KUKA KRL program: EPS_2_251455_MH61A_A_20251003045103.src

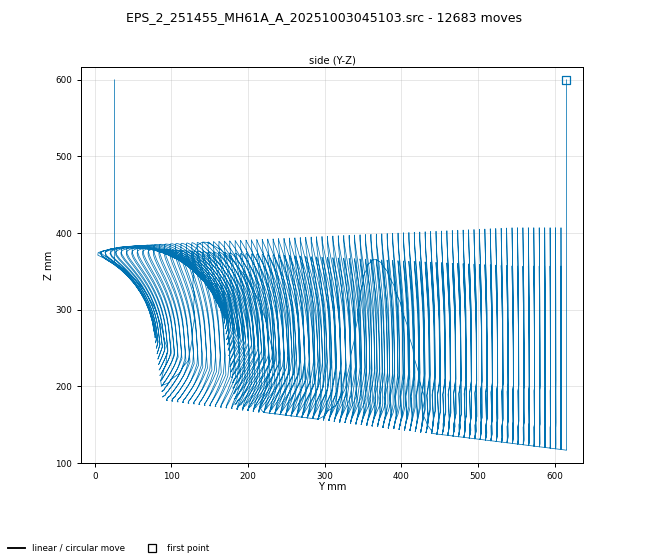
[picture p0: tool path of EPS_2_251455_MH61A_A_20251003045103.src, 12683 of 12685 moves have a stored position in this frame; points joined in program order, loops and branches not executed]
&ACCESS RVP
&REL 4
&COMMENT QRS 19112012
&PARAM EDITMASK = *
DEF PART()
EXT BAS (BAS_COMMAND :IN,REAL :IN )
INT I
BAS (#INITMOV,0 )

;KUKA QRS Post kuka4.cps  Date:22-06-2017 !

File_ID=2871

QRS_PRE_INIT()

;Init var - Until changes are made in qrs_pre_init
Outlet_Square_prg=0
Inlet_1_Square_prg=0
Inlet_2_Square_prg=0
Inlet_3_Square_prg=0
Inlet_4_Square_prg=0
Inlet_5_Square_prg=0

Outlet_1={X 0.000, Y 546.330, Z 306.500, B 0.000, E1 0.000 }
Inlet_1={X 0.000, Y 549.890, Z 256.500, B 0.000, E1 200.000 }
Outlet_1_type=201
Inlet_1_type=201
;QRS#1=Sidecore dimensions
;QRS#2=200-8" PVC SDR 35
;QRS#3=200-8" PVC SDR 35
;QRS#4=
;QRS#5=
;QRS#6=
;QRS#7=
;QRS#8=
;QRS#9=12-08 PSX
;QRS#10=12-08 PSX
;QRS#11=
;QRS#12=
;QRS#13=
;QRS#14=
;QRS#15=
;QRS#16=1220x127x686 2,25'
;QRS#17=EPS Height
;QRS#18=407
;QRS#19=*
;QRS#20= UPDATED VERSION 22-06-2017
;QRS#21=*
Outlet_Square=0100
Inlet_1_Square=0100
Inlet_2_Square=0
Inlet_3_Square=0
Inlet_4_Square=0
Inlet_5_Square=0
Mill_Square=1
Outlet_Square_Prg=204
Inlet_1_Square_prg=204

QRS_INIT()

$ADVANCE=5

; T1
PTP {E1 173.605,E2 173.605}
PTP {X 0,Y 615.512,A -85,B 0,C 180,E1 173.605,E2 173.605,E3 0,E4 0,E5 0,E6 0}
QRS_SPEED_INIT()
LIN {X 0,Y 615.512,Z 600,A -85,B 0,C 180,E1 173.605,E2 173.605,E3 0,E4 0,E5 0,E6 0} C_VEL
LIN {X 0,Y 615.512,Z 126.872,A -85,B 0,C 180,E1 173.605,E2 173.605} C_VEL
LIN {X 0,Y 615.512,Z 118.701,A -85,B 0,C 180,E1 173.605,E2 173.605} C_VEL
LIN {X 0,Y 615.489,Z 116.701,A -85,B 0,C 180,E1 173.42,E2 173.42} C_VEL
LIN {X 0,Y 615.462,Z 116.69,A -85,B 0,C 180,E1 170.801,E2 170.801} C_VEL
LIN {X 0,Y 615.487,Z 116.687,A -85,B 0,C 180,E1 168.139,E2 168.139} C_VEL
LIN {X 0,Y 615.481,Z 116.697,A -85,B 0,C 180,E1 165.451,E2 165.451} C_VEL
LIN {X 0,Y 615.47,Z 116.687,A -85,B 0,C 180,E1 162.729,E2 162.729} C_VEL
LIN {X 0,Y 615.49,Z 116.695,A -85,B 0,C 180,E1 159.967,E2 159.967} C_VEL
LIN {X 0,Y 615.479,Z 116.699,A -85,B 0,C 180,E1 157.656,E2 157.656} C_VEL
LIN {X 0,Y 615.464,Z 116.688,A -85,B 0,C 180,E1 155.007,E2 155.007} C_VEL
LIN {X 0,Y 615.489,Z 116.698,A -85,B 0,C 180,E1 152.085,E2 152.085} C_VEL
LIN {X 0,Y 615.484,Z 116.698,A -85,B 0,C 180,E1 149.84,E2 149.84} C_VEL
LIN {X 0,Y 615.463,Z 116.693,A -85,B 0,C 180,E1 147.541,E2 147.541} C_VEL
LIN {X 0,Y 615.466,Z 116.688,A -85,B 0,C 180,E1 145.184,E2 145.184} C_VEL
LIN {X 0,Y 615.495,Z 116.684,A -85,B 0,C 180,E1 142.758,E2 142.758} C_VEL
LIN {X 0,Y 615.472,Z 116.696,A -85,B 0,C 180,E1 139.913,E2 139.913} C_VEL
LIN {X 0,Y 615.458,Z 116.692,A -85,B 0,C 180,E1 137.645,E2 137.645} C_VEL
LIN {X 0,Y 615.496,Z 116.684,A -85,B 0,C 180,E1 134.932,E2 134.932} C_VEL
LIN {X 0,Y 615.471,Z 116.696,A -85,B 0,C 180,E1 132.079,E2 132.079} C_VEL
LIN {X 0,Y 615.459,Z 116.691,A -85,B 0,C 180,E1 129.752,E2 129.752} C_VEL
LIN {X 0,Y 615.491,Z 116.689,A -85,B 0,C 180,E1 126.937,E2 126.937} C_VEL
LIN {X 0,Y 615.459,Z 116.693,A -85,B 0,C 180,E1 124.024,E2 124.024} C_VEL
LIN {X 0,Y 615.464,Z 116.688,A -85,B 0,C 180,E1 121.687,E2 121.687} C_VEL
LIN {X 0,Y 615.486,Z 116.685,A -85,B 0,C 180,E1 119.406,E2 119.406} C_VEL
LIN {X 0,Y 615.471,Z 116.696,A -85,B 0,C 180,E1 116.445,E2 116.445} C_VEL
LIN {X 0,Y 615.461,Z 116.689,A -85,B 0,C 180,E1 114.003,E2 114.003} C_VEL
LIN {X 0,Y 615.496,Z 116.685,A -85,B 0,C 180,E1 111.431,E2 111.431} C_VEL
LIN {X 0,Y 615.469,Z 116.696,A -85,B 0,C 180,E1 108.6,E2 108.6} C_VEL
LIN {X 0,Y 615.475,Z 116.686,A -85,B 0,C 180,E1 105.905,E2 105.905} C_VEL
LIN {X 0,Y 615.491,Z 116.697,A -85,B 0,C 180,E1 103.201,E2 103.201} C_VEL
LIN {X 0,Y 615.46,Z 116.692,A -85,B 0,C 180,E1 100.527,E2 100.527} C_VEL
LIN {X 0,Y 615.485,Z 116.685,A -85,B 0,C 180,E1 97.876,E2 97.876} C_VEL
LIN {X 0,Y 615.494,Z 116.701,A -85,B 0,C 180,E1 95.241,E2 95.241} C_VEL
LIN {X 0,Y 615.459,Z 116.691,A -85,B 0,C 180,E1 92.618,E2 92.618} C_VEL
LIN {X 0,Y 615.486,Z 116.686,A -85,B 0,C 180,E1 90,E2 90} C_VEL
LIN {X 0,Y 615.496,Z 116.879,A -85,B 0,C 180,E1 87.955,E2 87.955} C_VEL
LIN {X 0,Y 615.461,Z 131.384,A -85,B 0,C 180,E1 85.415,E2 85.415} C_VEL
LIN {X 0,Y 615.445,Z 146.098,A -85,B 0,C 180,E1 82.866,E2 82.866} C_VEL
LIN {X 0,Y 615.45,Z 146.551,A -85,B 0,C 180,E1 82.804,E2 82.804} C_VEL
LIN {X 0,Y 615.45,Z 252.819,A -85,B 0,C 180,E1 81.545,E2 81.545} C_VEL
LIN {X 0,Y 615.452,Z 266.001,A -85,B 0,C 180,E1 81.256,E2 81.256} C_VEL
LIN {X 0,Y 615.481,Z 278.61,A -85,B 0,C 180,E1 80.842,E2 80.842} C_VEL
LIN {X 0,Y 615.493,Z 290.7,A -85,B 0,C 180,E1 80.304,E2 80.304} C_VEL
LIN {X 0,Y 615.485,Z 302.179,A -85,B 0,C 180,E1 79.639,E2 79.639} C_VEL
LIN {X 0,Y 615.499,Z 311.681,A -85,B 0,C 180,E1 78.957,E2 78.957} C_VEL
LIN {X 0,Y 615.497,Z 321.042,A -85,B 0,C 180,E1 78.139,E2 78.139} C_VEL
LIN {X 0,Y 615.498,Z 330.259,A -85,B 0,C 180,E1 77.135,E2 77.135} C_VEL
LIN {X 0,Y 615.496,Z 338.117,A -85,B 0,C 180,E1 76.064,E2 76.064} C_VEL
LIN {X 0,Y 615.497,Z 343.66,A -85,B 0,C 180,E1 75.113,E2 75.113} C_VEL
LIN {X 0,Y 615.492,Z 348.346,A -85,B 0,C 180,E1 74.095,E2 74.095} C_VEL
LIN {X 0,Y 615.495,Z 351.892,A -85,B 0,C 180,E1 73.072,E2 73.072} C_VEL
LIN {X 0,Y 615.498,Z 354.389,A -85,B 0,C 180,E1 72.043,E2 72.043} C_VEL
LIN {X 0,Y 615.494,Z 355.474,A -85,B 0,C 180,E1 71.354,E2 71.354} C_VEL
LIN {X 0,Y 615.496,Z 356.136,A -85,B 0,C 180,E1 70.662,E2 70.662} C_VEL
LIN {X 0,Y 615.497,Z 356.267,A -85,B 0,C 180,E1 69.441,E2 69.441} C_VEL
LIN {X 0,Y 615.498,Z 355.487,A -85,B 0,C 180,E1 68.568,E2 68.568} C_VEL
LIN {X 0,Y 615.492,Z 353.93,A -85,B 0,C 180,E1 67.653,E2 67.653} C_VEL
LIN {X 0,Y 615.496,Z 350.636,A -85,B 0,C 180,E1 66.444,E2 66.444} C_VEL
LIN {X 0,Y 615.495,Z 346.435,A -85,B 0,C 180,E1 65.369,E2 65.369} C_VEL
LIN {X 0,Y 615.494,Z 340.815,A -85,B 0,C 180,E1 64.284,E2 64.284} C_VEL
LIN {X 0,Y 615.498,Z 334,A -85,B 0,C 180,E1 63.255,E2 63.255} C_VEL
LIN {X 0,Y 615.499,Z 325.884,A -85,B 0,C 180,E1 62.27,E2 62.27} C_VEL
LIN {X 0,Y 615.497,Z 317.556,A -85,B 0,C 180,E1 61.445,E2 61.445} C_VEL
LIN {X 0,Y 615.498,Z 306.914,A -85,B 0,C 180,E1 60.594,E2 60.594} C_VEL
LIN {X 0,Y 615.46,Z 296.655,A -85,B 0,C 180,E1 59.931,E2 59.931} C_VEL
LIN {X 0,Y 615.489,Z 284.671,A -85,B 0,C 180,E1 59.318,E2 59.318} C_VEL
LIN {X 0,Y 615.495,Z 272.133,A -85,B 0,C 180,E1 58.838,E2 58.838} C_VEL
LIN {X 0,Y 615.481,Z 259.797,A -85,B 0,C 180,E1 58.501,E2 58.501} C_VEL
LIN {X 0,Y 615.471,Z 246.219,A -85,B 0,C 180,E1 58.273,E2 58.273} C_VEL
LIN {X 0,Y 615.485,Z 146.442,A -85,B 0,C 180,E1 57.105,E2 57.105} C_VEL
LIN {X 0,Y 615.488,Z 129.487,A -85,B 0,C 180,E1 54.166,E2 54.166} C_VEL
LIN {X 0,Y 615.444,Z 116.696,A -85,B 0,C 180,E1 51.902,E2 51.902} C_VEL
LIN {X 0,Y 615.449,Z 116.693,A -85,B 0,C 180,E1 49.39,E2 49.39} C_VEL
LIN {X 0,Y 615.498,Z 116.697,A -85,B 0,C 180,E1 46.756,E2 46.756} C_VEL
LIN {X 0,Y 615.441,Z 116.697,A -85,B 0,C 180,E1 44.154,E2 44.154} C_VEL
LIN {X 0,Y 615.434,Z 116.697,A -85,B 0,C 180,E1 42.074,E2 42.074} C_VEL
LIN {X 0,Y 615.434,Z 116.695,A -85,B 0,C 180,E1 39.754,E2 39.754} C_VEL
LIN {X 0,Y 615.487,Z 116.694,A -85,B 0,C 180,E1 37.242,E2 37.242} C_VEL
LIN {X 0,Y 615.455,Z 116.699,A -85,B 0,C 180,E1 34.696,E2 34.696} C_VEL
LIN {X 0,Y 615.427,Z 116.698,A -85,B 0,C 180,E1 32.322,E2 32.322} C_VEL
LIN {X 0,Y 615.444,Z 116.696,A -85,B 0,C 180,E1 29.787,E2 29.787} C_VEL
LIN {X 0,Y 615.466,Z 116.7,A -85,B 0,C 180,E1 27.041,E2 27.041} C_VEL
LIN {X 0,Y 615.452,Z 116.699,A -85,B 0,C 180,E1 24.993,E2 24.993} C_VEL
LIN {X 0,Y 615.431,Z 116.7,A -85,B 0,C 180,E1 22.847,E2 22.847} C_VEL
LIN {X 0,Y 615.417,Z 116.699,A -85,B 0,C 180,E1 20.539,E2 20.539} C_VEL
LIN {X 0,Y 615.449,Z 116.699,A -85,B 0,C 180,E1 17.958,E2 17.958} C_VEL
LIN {X 0,Y 615.442,Z 116.7,A -85,B 0,C 180,E1 15.227,E2 15.227} C_VEL
LIN {X 0,Y 615.434,Z 116.7,A -85,B 0,C 180,E1 13.202,E2 13.202} C_VEL
LIN {X 0,Y 615.415,Z 116.7,A -85,B 0,C 180,E1 10.852,E2 10.852} C_VEL
LIN {X 0,Y 615.424,Z 116.7,A -85,B 0,C 180,E1 8.537,E2 8.537} C_VEL
LIN {X 0,Y 615.498,Z 116.699,A -85,B 0,C 180,E1 5.898,E2 5.898} C_VEL
LIN {X 0,Y 615.428,Z 116.698,A -85,B 0,C 180,E1 3.273,E2 3.273} C_VEL
LIN {X 0,Y 615.428,Z 116.698,A -85,B 0,C 180,E1 1.309,E2 1.309} C_VEL
LIN {X 0,Y 615.429,Z 116.697,A -85,B 0,C 180,E1 -0.654,E2 -0.654} C_VEL
LIN {X 0,Y 615.429,Z 116.697,A -85,B 0,C 180,E1 -2.618,E2 -2.618} C_VEL
LIN {X 0,Y 615.43,Z 116.696,A -85,B 0,C 180,E1 -4.585,E2 -4.585} C_VEL
LIN {X 0,Y 615.431,Z 116.696,A -85,B 0,C 180,E1 -6.557,E2 -6.557} C_VEL
LIN {X 0,Y 615.431,Z 116.696,A -85,B 0,C 180,E1 -8.538,E2 -8.538} C_VEL
LIN {X 0,Y 615.434,Z 116.697,A -85,B 0,C 180,E1 -10.861,E2 -10.861} C_VEL
LIN {X 0,Y 615.465,Z 116.699,A -85,B 0,C 180,E1 -13.202,E2 -13.202} C_VEL
LIN {X 0,Y 615.467,Z 116.692,A -85,B 0,C 180,E1 -15.906,E2 -15.906} C_VEL
LIN {X 0,Y 615.457,Z 116.693,A -85,B 0,C 180,E1 -17.958,E2 -17.958} C_VEL
LIN {X 0,Y 615.439,Z 116.696,A -85,B 0,C 180,E1 -20.544,E2 -20.544} C_VEL
LIN {X 0,Y 615.462,Z 116.698,A -85,B 0,C 180,E1 -22.846,E2 -22.846} C_VEL
LIN {X 0,Y 615.466,Z 116.691,A -85,B 0,C 180,E1 -25.717,E2 -25.717} C_VEL
LIN {X 0,Y 615.448,Z 116.692,A -85,B 0,C 180,E1 -27.917,E2 -27.917} C_VEL
LIN {X 0,Y 615.443,Z 116.694,A -85,B 0,C 180,E1 -30.163,E2 -30.163} C_VEL
LIN {X 0,Y 615.458,Z 116.697,A -85,B 0,C 180,E1 -32.459,E2 -32.459} C_VEL
LIN {X 0,Y 615.499,Z 116.7,A -85,B 0,C 180,E1 -34.815,E2 -34.815} C_VEL
LIN {X 0,Y 615.489,Z 116.687,A -85,B 0,C 180,E1 -37.242,E2 -37.242} C_VEL
LIN {X 0,Y 615.448,Z 116.692,A -85,B 0,C 180,E1 -39.753,E2 -39.753} C_VEL
LIN {X 0,Y 615.477,Z 116.698,A -85,B 0,C 180,E1 -42.354,E2 -42.354} C_VEL
LIN {X 0,Y 615.492,Z 116.685,A -85,B 0,C 180,E1 -45.068,E2 -45.068} C_VEL
LIN {X 0,Y 615.453,Z 116.692,A -85,B 0,C 180,E1 -47.644,E2 -47.644} C_VEL
LIN {X 0,Y 615.493,Z 116.699,A -85,B 0,C 180,E1 -50.25,E2 -50.25} C_VEL
LIN {X 0,Y 615.475,Z 116.686,A -85,B 0,C 180,E1 -53.065,E2 -53.065} C_VEL
LIN {X 0,Y 615.46,Z 116.69,A -85,B 0,C 180,E1 -55.303,E2 -55.303} C_VEL
LIN {X 0,Y 615.464,Z 116.695,A -85,B 0,C 180,E1 -57.673,E2 -57.673} C_VEL
LIN {X 0,Y 615.489,Z 116.686,A -85,B 0,C 180,E1 -60.594,E2 -60.594} C_VEL
LIN {X 0,Y 615.468,Z 116.687,A -85,B 0,C 180,E1 -62.959,E2 -62.959} C_VEL
LIN {X 0,Y 615.485,Z 116.7,A -85,B 0,C 180,E1 -65.728,E2 -65.728} C_VEL
LIN {X 0,Y 615.464,Z 116.822,A -85,B 0,C 180,E1 -67.066,E2 -67.066} C_VEL
LIN {X 0,Y 615.465,Z 136.77,A -85,B 0,C 180,E1 -69.706,E2 -69.706} C_VEL
LIN {X 0,Y 615.485,Z 158.669,A -85,B 0,C 180,E1 -72.558,E2 -72.558} C_VEL
LIN {X 0,Y 615.469,Z 179.891,A -85,B 0,C 180,E1 -75.281,E2 -75.281} C_VEL
LIN {X 0,Y 615.452,Z 194.3,A -85,B 0,C 180,E1 -77.113,E2 -77.113} C_VEL
LIN {X 0,Y 615.488,Z 302.823,A -85,B 0,C 180,E1 -78.411,E2 -78.411} C_VEL
LIN {X 0,Y 615.477,Z 315.341,A -85,B 0,C 180,E1 -78.682,E2 -78.682} C_VEL
LIN {X 0,Y 615.488,Z 328.618,A -85,B 0,C 180,E1 -79.113,E2 -79.113} C_VEL
LIN {X 0,Y 615.477,Z 340.476,A -85,B 0,C 180,E1 -79.639,E2 -79.639} C_VEL
LIN {X 0,Y 615.494,Z 351.992,A -85,B 0,C 180,E1 -80.304,E2 -80.304} C_VEL
LIN {X 0,Y 615.499,Z 362.339,A -85,B 0,C 180,E1 -81.05,E2 -81.05} C_VEL
LIN {X 0,Y 615.497,Z 370.81,A -85,B 0,C 180,E1 -81.794,E2 -81.794} C_VEL
LIN {X 0,Y 615.498,Z 378.605,A -85,B 0,C 180,E1 -82.619,E2 -82.619} C_VEL
LIN {X 0,Y 615.496,Z 386.202,A -85,B 0,C 180,E1 -83.608,E2 -83.608} C_VEL
LIN {X 0,Y 615.498,Z 393.204,A -85,B 0,C 180,E1 -84.759,E2 -84.759} C_VEL
LIN {X 0,Y 615.494,Z 397.851,A -85,B 0,C 180,E1 -85.743,E2 -85.743} C_VEL
LIN {X 0,Y 615.494,Z 401.398,A -85,B 0,C 180,E1 -86.727,E2 -86.727} C_VEL
LIN {X 0,Y 615.497,Z 403.233,A -85,B 0,C 180,E1 -87.382,E2 -87.382} C_VEL
LIN {X 0,Y 615.5,Z 404.607,A -85,B 0,C 180,E1 -88.037,E2 -88.037} C_VEL
LIN {X 0,Y 615.496,Z 406.173,A -85,B 0,C 180,E1 -89.346,E2 -89.346} C_VEL
LIN {X 0,Y 615.494,Z 406.389,A -85,B 0,C 180,E1 -90,E2 -90} C_VEL
LIN {X 0,Y 615.495,Z 405.58,A -85,B 0,C 180,E1 -91.308,E2 -91.308} C_VEL
LIN {X 0,Y 615.5,Z 404.608,A -85,B 0,C 180,E1 -91.963,E2 -91.963} C_VEL
LIN {X 0,Y 615.497,Z 403.233,A -85,B 0,C 180,E1 -92.618,E2 -92.618} C_VEL
LIN {X 0,Y 615.496,Z 400.35,A -85,B 0,C 180,E1 -93.601,E2 -93.601} C_VEL
LIN {X 0,Y 615.498,Z 396.442,A -85,B 0,C 180,E1 -94.584,E2 -94.584} C_VEL
LIN {X 0,Y 615.499,Z 391.405,A -85,B 0,C 180,E1 -95.57,E2 -95.57} C_VEL
LIN {X 0,Y 615.497,Z 384.87,A -85,B 0,C 180,E1 -96.583,E2 -96.583} C_VEL
LIN {X 0,Y 615.497,Z 377.134,A -85,B 0,C 180,E1 -97.545,E2 -97.545} C_VEL
LIN {X 0,Y 615.498,Z 369.046,A -85,B 0,C 180,E1 -98.371,E2 -98.371} C_VEL
LIN {X 0,Y 615.499,Z 359.169,A -85,B 0,C 180,E1 -99.198,E2 -99.198} C_VEL
LIN {X 0,Y 615.488,Z 347.983,A -85,B 0,C 180,E1 -99.945,E2 -99.945} C_VEL
LIN {X 0,Y 615.482,Z 337.026,A -85,B 0,C 180,E1 -100.527,E2 -100.527} C_VEL
LIN {X 0,Y 615.48,Z 324.492,A -85,B 0,C 180,E1 -101.04,E2 -101.04} C_VEL
LIN {X 0,Y 615.479,Z 312.072,A -85,B 0,C 180,E1 -101.402,E2 -101.402} C_VEL
LIN {X 0,Y 615.493,Z 298.473,A -85,B 0,C 180,E1 -101.652,E2 -101.652} C_VEL
LIN {X 0,Y 615.452,Z 194.302,A -85,B 0,C 180,E1 -102.887,E2 -102.887} C_VEL
LIN {X 0,Y 615.494,Z 171.934,A -85,B 0,C 180,E1 -105.735,E2 -105.735} C_VEL
LIN {X 0,Y 615.456,Z 151.013,A -85,B 0,C 180,E1 -108.435,E2 -108.435} C_VEL
LIN {X 0,Y 615.488,Z 130.783,A -85,B 0,C 180,E1 -111.081,E2 -111.081} C_VEL
LIN {X 0,Y 615.465,Z 116.689,A -85,B 0,C 180,E1 -112.978,E2 -112.978} C_VEL
LIN {X 0,Y 615.489,Z 116.689,A -85,B 0,C 180,E1 -115.716,E2 -115.716} C_VEL
LIN {X 0,Y 615.469,Z 116.695,A -85,B 0,C 180,E1 -118.447,E2 -118.447} C_VEL
LIN {X 0,Y 615.479,Z 116.685,A -85,B 0,C 180,E1 -121.084,E2 -121.084} C_VEL
LIN {X 0,Y 615.49,Z 116.7,A -85,B 0,C 180,E1 -124.022,E2 -124.022} C_VEL
LIN {X 0,Y 615.477,Z 116.685,A -85,B 0,C 180,E1 -126.935,E2 -126.935} C_VEL
LIN {X 0,Y 615.493,Z 116.699,A -85,B 0,C 180,E1 -129.75,E2 -129.75} C_VEL
LIN {X 0,Y 615.464,Z 116.692,A -85,B 0,C 180,E1 -132.355,E2 -132.355} C_VEL
LIN {X 0,Y 615.492,Z 116.684,A -85,B 0,C 180,E1 -135.068,E2 -135.068} C_VEL
LIN {X 0,Y 615.475,Z 116.696,A -85,B 0,C 180,E1 -137.921,E2 -137.921} C_VEL
LIN {X 0,Y 615.462,Z 116.691,A -85,B 0,C 180,E1 -140.248,E2 -140.248} C_VEL
LIN {X 0,Y 615.49,Z 116.688,A -85,B 0,C 180,E1 -143.063,E2 -143.063} C_VEL
LIN {X 0,Y 615.464,Z 116.693,A -85,B 0,C 180,E1 -145.976,E2 -145.976} C_VEL
LIN {X 0,Y 615.466,Z 116.688,A -85,B 0,C 180,E1 -148.313,E2 -148.313} C_VEL
LIN {X 0,Y 615.486,Z 116.684,A -85,B 0,C 180,E1 -150.593,E2 -150.593} C_VEL
LIN {X 0,Y 615.472,Z 116.697,A -85,B 0,C 180,E1 -153.555,E2 -153.555} C_VEL
LIN {X 0,Y 615.464,Z 116.689,A -85,B 0,C 180,E1 -155.996,E2 -155.996} C_VEL
LIN {X 0,Y 615.495,Z 116.684,A -85,B 0,C 180,E1 -158.568,E2 -158.568} C_VEL
LIN {X 0,Y 615.474,Z 116.696,A -85,B 0,C 180,E1 -161.399,E2 -161.399} C_VEL
LIN {X 0,Y 615.476,Z 116.685,A -85,B 0,C 180,E1 -164.094,E2 -164.094} C_VEL
LIN {X 0,Y 615.49,Z 116.695,A -85,B 0,C 180,E1 -166.799,E2 -166.799} C_VEL
LIN {X 0,Y 615.462,Z 116.693,A -85,B 0,C 180,E1 -169.472,E2 -169.472} C_VEL
LIN {X 0,Y 615.485,Z 116.685,A -85,B 0,C 180,E1 -172.124,E2 -172.124} C_VEL
LIN {X 0,Y 615.492,Z 116.7,A -85,B 0,C 180,E1 -174.759,E2 -174.759} C_VEL
LIN {X 0,Y 615.462,Z 116.691,A -85,B 0,C 180,E1 -177.382,E2 -177.382} C_VEL
LIN {X 0,Y 615.486,Z 116.685,A -85,B 0,C 180,E1 -180,E2 -180} C_VEL
LIN {X 0,Y 615.492,Z 116.702,A -85,B 0,C 180,E1 -182.618,E2 -182.618} C_VEL
LIN {X 0,Y 615.457,Z 116.692,A -85,B 0,C 180,E1 -185.241,E2 -185.241} C_VEL
LIN {X 0,Y 615.489,Z 116.701,A -85,B 0,C 180,E1 -186.58,E2 -186.58} C_VEL
LIN {X 0,Y 614.793,Z 116.838,A -85,B 0,C 180,E1 -187.126,E2 -187.126} C_VEL
LIN {X 0,Y 611.942,Z 117.256,A -85,B 0,C 180,E1 -188.012,E2 -188.012} C_VEL
LIN {X 0,Y 609.554,Z 117.563,A -85,B 0,C 180,E1 -188.725,E2 -188.725} C_VEL
LIN {X 0,Y 608.531,Z 117.679,A -85,B 0,C 180,E1 -189.274,E2 -189.274} C_VEL
LIN {X 0,Y 608.448,Z 117.688,A -85,B 0,C 180,E1 -189.461,E2 -189.461} C_VEL
LIN {X 0,Y 608.462,Z 117.69,A -85,B 0,C 180,E1 -192,E2 -192} C_VEL
LIN {X 0,Y 608.467,Z 117.69,A -85,B 0,C 180,E1 -194.721,E2 -194.721} C_VEL
LIN {X 0,Y 608.443,Z 117.689,A -85,B 0,C 180,E1 -197.477,E2 -197.477} C_VEL
LIN {X 0,Y 608.458,Z 117.697,A -85,B 0,C 180,E1 -200.274,E2 -200.274} C_VEL
LIN {X 0,Y 608.458,Z 117.692,A -85,B 0,C 180,E1 -202.476,E2 -202.476} C_VEL
LIN {X 0,Y 608.444,Z 117.692,A -85,B 0,C 180,E1 -204.571,E2 -204.571} C_VEL
LIN {X 0,Y 608.47,Z 117.686,A -85,B 0,C 180,E1 -207.206,E2 -207.206} C_VEL
LIN {X 0,Y 608.47,Z 117.696,A -85,B 0,C 180,E1 -209.972,E2 -209.972} C_VEL
LIN {X 0,Y 608.449,Z 117.688,A -85,B 0,C 180,E1 -212.88,E2 -212.88} C_VEL
LIN {X 0,Y 608.438,Z 117.691,A -85,B 0,C 180,E1 -215.278,E2 -215.278} C_VEL
LIN {X 0,Y 608.466,Z 117.695,A -85,B 0,C 180,E1 -217.746,E2 -217.746} C_VEL
LIN {X 0,Y 608.433,Z 117.692,A -85,B 0,C 180,E1 -220.327,E2 -220.327} C_VEL
LIN {X 0,Y 608.451,Z 117.688,A -85,B 0,C 180,E1 -222.96,E2 -222.96} C_VEL
LIN {X 0,Y 608.451,Z 117.697,A -85,B 0,C 180,E1 -225.737,E2 -225.737} C_VEL
LIN {X 0,Y 608.452,Z 117.688,A -85,B 0,C 180,E1 -228.659,E2 -228.659} C_VEL
LIN {X 0,Y 608.453,Z 117.694,A -85,B 0,C 180,E1 -231.761,E2 -231.761} C_VEL
LIN {X 0,Y 608.438,Z 117.692,A -85,B 0,C 180,E1 -233.956,E2 -233.956} C_VEL
LIN {X 0,Y 608.442,Z 117.689,A -85,B 0,C 180,E1 -236.328,E2 -236.328} C_VEL
LIN {X 0,Y 608.448,Z 117.69,A -85,B 0,C 180,E1 -238.732,E2 -238.732} C_VEL
LIN {X 0,Y 608.469,Z 117.695,A -85,B 0,C 180,E1 -241.381,E2 -241.381} C_VEL
LIN {X 0,Y 608.432,Z 117.691,A -85,B 0,C 180,E1 -243.964,E2 -243.964} C_VEL
LIN {X 0,Y 608.451,Z 117.693,A -85,B 0,C 180,E1 -246.876,E2 -246.876} C_VEL
LIN {X 0,Y 608.457,Z 117.694,A -85,B 0,C 180,E1 -249.324,E2 -249.324} C_VEL
LIN {X 0,Y 608.432,Z 117.691,A -85,B 0,C 180,E1 -251.828,E2 -251.828} C_VEL
LIN {X 0,Y 608.472,Z 117.689,A -85,B 0,C 180,E1 -254.594,E2 -254.594} C_VEL
LIN {X 0,Y 608.459,Z 117.691,A -85,B 0,C 180,E1 -257.323,E2 -257.323} C_VEL
LIN {X 0,Y 608.456,Z 117.687,A -85,B 0,C 180,E1 -260.023,E2 -260.023} C_VEL
LIN {X 0,Y 608.466,Z 117.695,A -85,B 0,C 180,E1 -262.701,E2 -262.701} C_VEL
LIN {X 0,Y 608.473,Z 117.695,A -85,B 0,C 180,E1 -264.698,E2 -264.698} C_VEL
LIN {X 0,Y 608.454,Z 117.689,A -85,B 0,C 180,E1 -267.352,E2 -267.352} C_VEL
LIN {X 0,Y 608.477,Z 117.686,A -85,B 0,C 180,E1 -270,E2 -270} C_VEL
LIN {X 0,Y 608.489,Z 117.837,A -85,B 0,C 180,E1 -271.986,E2 -271.986} C_VEL
LIN {X 0,Y 608.429,Z 132.862,A -85,B 0,C 180,E1 -274.638,E2 -274.638} C_VEL
LIN {X 0,Y 608.412,Z 146.625,A -85,B 0,C 180,E1 -277.039,E2 -277.039} C_VEL
LIN {X 0,Y 608.499,Z 253.014,A -85,B 0,C 180,E1 -278.322,E2 -278.322} C_VEL
LIN {X 0,Y 608.512,Z 266.142,A -85,B 0,C 180,E1 -278.614,E2 -278.614} C_VEL
LIN {X 0,Y 608.503,Z 279.349,A -85,B 0,C 180,E1 -279.054,E2 -279.054} C_VEL
LIN {X 0,Y 608.521,Z 290.485,A -85,B 0,C 180,E1 -279.557,E2 -279.557} C_VEL
LIN {X 0,Y 608.476,Z 302.094,A -85,B 0,C 180,E1 -280.229,E2 -280.229} C_VEL
LIN {X 0,Y 608.49,Z 313.195,A -85,B 0,C 180,E1 -281.038,E2 -281.038} C_VEL
LIN {X 0,Y 608.463,Z 322.009,A -85,B 0,C 180,E1 -281.831,E2 -281.831} C_VEL
LIN {X 0,Y 608.47,Z 331.155,A -85,B 0,C 180,E1 -282.847,E2 -282.847} C_VEL
LIN {X 0,Y 608.448,Z 338.761,A -85,B 0,C 180,E1 -283.898,E2 -283.898} C_VEL
LIN {X 0,Y 608.439,Z 345.31,A -85,B 0,C 180,E1 -285.064,E2 -285.064} C_VEL
LIN {X 0,Y 608.431,Z 349.765,A -85,B 0,C 180,E1 -286.095,E2 -286.095} C_VEL
LIN {X 0,Y 608.428,Z 352.118,A -85,B 0,C 180,E1 -286.785,E2 -286.785} C_VEL
LIN {X 0,Y 608.421,Z 353.999,A -85,B 0,C 180,E1 -287.478,E2 -287.478} C_VEL
LIN {X 0,Y 608.428,Z 356.164,A -85,B 0,C 180,E1 -288.704,E2 -288.704} C_VEL
LIN {X 0,Y 608.419,Z 356.895,A -85,B 0,C 180,E1 -289.572,E2 -289.572} C_VEL
LIN {X 0,Y 608.441,Z 356.808,A -85,B 0,C 180,E1 -290.672,E2 -290.672} C_VEL
LIN {X 0,Y 608.42,Z 355.762,A -85,B 0,C 180,E1 -291.694,E2 -291.694} C_VEL
LIN {X 0,Y 608.429,Z 354.308,A -85,B 0,C 180,E1 -292.47,E2 -292.47} C_VEL
LIN {X 0,Y 608.426,Z 351.543,A -85,B 0,C 180,E1 -293.485,E2 -293.485} C_VEL
LIN {X 0,Y 608.426,Z 347.423,A -85,B 0,C 180,E1 -294.572,E2 -294.572} C_VEL
LIN {X 0,Y 608.435,Z 341.672,A -85,B 0,C 180,E1 -295.714,E2 -295.714} C_VEL
LIN {X 0,Y 608.444,Z 334.754,A -85,B 0,C 180,E1 -296.775,E2 -296.775} C_VEL
LIN {X 0,Y 608.48,Z 327.251,A -85,B 0,C 180,E1 -297.703,E2 -297.703} C_VEL
LIN {X 0,Y 608.482,Z 318.186,A -85,B 0,C 180,E1 -298.622,E2 -298.622} C_VEL
LIN {X 0,Y 608.486,Z 308.754,A -85,B 0,C 180,E1 -299.398,E2 -299.398} C_VEL
LIN {X 0,Y 608.466,Z 297.58,A -85,B 0,C 180,E1 -300.141,E2 -300.141} C_VEL
LIN {X 0,Y 608.504,Z 285.303,A -85,B 0,C 180,E1 -300.784,E2 -300.784} C_VEL
LIN {X 0,Y 608.525,Z 273.681,A -85,B 0,C 180,E1 -301.244,E2 -301.244} C_VEL
LIN {X 0,Y 608.527,Z 260.033,A -85,B 0,C 180,E1 -301.628,E2 -301.628} C_VEL
LIN {X 0,Y 608.545,Z 246.638,A -85,B 0,C 180,E1 -301.858,E2 -301.858} C_VEL
LIN {X 0,Y 608.472,Z 146.615,A -85,B 0,C 180,E1 -303.051,E2 -303.051} C_VEL
LIN {X 0,Y 608.473,Z 130.557,A -85,B 0,C 180,E1 -305.856,E2 -305.856} C_VEL
LIN {X 0,Y 608.42,Z 117.694,A -85,B 0,C 180,E1 -308.141,E2 -308.141} C_VEL
LIN {X 0,Y 608.433,Z 117.69,A -85,B 0,C 180,E1 -310.327,E2 -310.327} C_VEL
LIN {X 0,Y 608.482,Z 117.695,A -85,B 0,C 180,E1 -313.31,E2 -313.31} C_VEL
LIN {X 0,Y 608.429,Z 117.691,A -85,B 0,C 180,E1 -316.127,E2 -316.127} C_VEL
LIN {X 0,Y 608.448,Z 117.693,A -85,B 0,C 180,E1 -318.823,E2 -318.823} C_VEL
LIN {X 0,Y 608.428,Z 117.692,A -85,B 0,C 180,E1 -321.765,E2 -321.765} C_VEL
LIN {X 0,Y 608.426,Z 117.691,A -85,B 0,C 180,E1 -323.957,E2 -323.957} C_VEL
LIN {X 0,Y 608.443,Z 117.691,A -85,B 0,C 180,E1 -326.328,E2 -326.328} C_VEL
LIN {X 0,Y 608.444,Z 117.697,A -85,B 0,C 180,E1 -328.733,E2 -328.733} C_VEL
LIN {X 0,Y 608.426,Z 117.693,A -85,B 0,C 180,E1 -331.389,E2 -331.389} C_VEL
LIN {X 0,Y 608.409,Z 117.696,A -85,B 0,C 180,E1 -333.224,E2 -333.224} C_VEL
LIN {X 0,Y 608.41,Z 117.693,A -85,B 0,C 180,E1 -335.427,E2 -335.427} C_VEL
LIN {X 0,Y 608.454,Z 117.694,A -85,B 0,C 180,E1 -338.308,E2 -338.308} C_VEL
LIN {X 0,Y 608.406,Z 117.694,A -85,B 0,C 180,E1 -341.303,E2 -341.303} C_VEL
LIN {X 0,Y 608.421,Z 117.695,A -85,B 0,C 180,E1 -343.905,E2 -343.905} C_VEL
LIN {X 0,Y 608.423,Z 117.696,A -85,B 0,C 180,E1 -346.643,E2 -346.643} C_VEL
LIN {X 0,Y 608.4,Z 117.694,A -85,B 0,C 180,E1 -349.349,E2 -349.349} C_VEL
LIN {X 0,Y 608.435,Z 117.699,A -85,B 0,C 180,E1 -352.033,E2 -352.033} C_VEL
LIN {X 0,Y 608.414,Z 117.694,A -85,B 0,C 180,E1 -354.698,E2 -354.698} C_VEL
LIN {X 0,Y 608.428,Z 117.692,A -85,B 0,C 180,E1 -357.352,E2 -357.352} C_VEL
LIN {X 0,Y 608.475,Z 117.693,A -85,B 0,C 180,E1 -360,E2 -360} C_VEL
LIN {X 0,Y 608.425,Z 117.691,A -85,B 0,C 180,E1 -362.648,E2 -362.648} C_VEL
LIN {X 0,Y 608.43,Z 117.694,A -85,B 0,C 180,E1 -365.302,E2 -365.302} C_VEL
LIN {X 0,Y 608.469,Z 117.69,A -85,B 0,C 180,E1 -367.967,E2 -367.967} C_VEL
LIN {X 0,Y 608.432,Z 117.692,A -85,B 0,C 180,E1 -370.937,E2 -370.937} C_VEL
LIN {X 0,Y 608.447,Z 117.697,A -85,B 0,C 180,E1 -373.357,E2 -373.357} C_VEL
LIN {X 0,Y 608.431,Z 117.691,A -85,B 0,C 180,E1 -376.095,E2 -376.095} C_VEL
LIN {X 0,Y 608.439,Z 117.693,A -85,B 0,C 180,E1 -378.87,E2 -378.87} C_VEL
LIN {X 0,Y 608.459,Z 117.689,A -85,B 0,C 180,E1 -381.692,E2 -381.692} C_VEL
LIN {X 0,Y 608.431,Z 117.693,A -85,B 0,C 180,E1 -384.572,E2 -384.572} C_VEL
LIN {X 0,Y 608.489,Z 117.69,A -85,B 0,C 180,E1 -387.209,E2 -387.209} C_VEL
LIN {X 0,Y 608.418,Z 117.692,A -85,B 0,C 180,E1 -389.963,E2 -389.963} C_VEL
LIN {X 0,Y 608.439,Z 117.694,A -85,B 0,C 180,E1 -392.519,E2 -392.519} C_VEL
LIN {X 0,Y 608.433,Z 117.693,A -85,B 0,C 180,E1 -395.279,E2 -395.279} C_VEL
LIN {X 0,Y 608.447,Z 117.688,A -85,B 0,C 180,E1 -397.748,E2 -397.748} C_VEL
LIN {X 0,Y 608.435,Z 117.695,A -85,B 0,C 180,E1 -400.327,E2 -400.327} C_VEL
LIN {X 0,Y 608.465,Z 117.687,A -85,B 0,C 180,E1 -403.308,E2 -403.308} C_VEL
LIN {X 0,Y 608.452,Z 117.693,A -85,B 0,C 180,E1 -406.129,E2 -406.129} C_VEL
LIN {X 0,Y 608.458,Z 117.69,A -85,B 0,C 180,E1 -408.824,E2 -408.824} C_VEL
LIN {X 0,Y 608.43,Z 117.691,A -85,B 0,C 180,E1 -411.409,E2 -411.409} C_VEL
LIN {X 0,Y 608.447,Z 117.695,A -85,B 0,C 180,E1 -413.955,E2 -413.955} C_VEL
LIN {X 0,Y 608.469,Z 117.693,A -85,B 0,C 180,E1 -416.329,E2 -416.329} C_VEL
LIN {X 0,Y 608.448,Z 117.689,A -85,B 0,C 180,E1 -418.733,E2 -418.733} C_VEL
LIN {X 0,Y 608.455,Z 117.689,A -85,B 0,C 180,E1 -421.384,E2 -421.384} C_VEL
LIN {X 0,Y 608.441,Z 117.699,A -85,B 0,C 180,E1 -423.964,E2 -423.964} C_VEL
LIN {X 0,Y 608.472,Z 117.692,A -85,B 0,C 180,E1 -426.155,E2 -426.155} C_VEL
LIN {X 0,Y 608.468,Z 117.819,A -85,B 0,C 180,E1 -426.922,E2 -426.922} C_VEL
LIN {X 0,Y 608.585,Z 133.442,A -85,B 0,C 180,E1 -429.023,E2 -429.023} C_VEL
LIN {X 0,Y 608.522,Z 154.715,A -85,B 0,C 180,E1 -431.83,E2 -431.83} C_VEL
LIN {X 0,Y 608.49,Z 175.989,A -85,B 0,C 180,E1 -434.594,E2 -434.594} C_VEL
LIN {X 0,Y 608.45,Z 194.521,A -85,B 0,C 180,E1 -436.972,E2 -436.972} C_VEL
LIN {X 0,Y 608.547,Z 302.94,A -85,B 0,C 180,E1 -438.276,E2 -438.276} C_VEL
LIN {X 0,Y 608.512,Z 316.212,A -85,B 0,C 180,E1 -438.571,E2 -438.571} C_VEL
LIN {X 0,Y 608.514,Z 328.628,A -85,B 0,C 180,E1 -438.982,E2 -438.982} C_VEL
LIN {X 0,Y 608.499,Z 340.632,A -85,B 0,C 180,E1 -439.519,E2 -439.519} C_VEL
LIN {X 0,Y 608.484,Z 352.195,A -85,B 0,C 180,E1 -440.191,E2 -440.191} C_VEL
LIN {X 0,Y 608.485,Z 362.592,A -85,B 0,C 180,E1 -440.946,E2 -440.946} C_VEL
LIN {X 0,Y 608.475,Z 371.11,A -85,B 0,C 180,E1 -441.699,E2 -441.699} C_VEL
LIN {X 0,Y 608.471,Z 378.959,A -85,B 0,C 180,E1 -442.534,E2 -442.534} C_VEL
LIN {X 0,Y 608.461,Z 386.286,A -85,B 0,C 180,E1 -443.484,E2 -443.484} C_VEL
LIN {X 0,Y 608.451,Z 391.865,A -85,B 0,C 180,E1 -444.365,E2 -444.365} C_VEL
LIN {X 0,Y 608.432,Z 396.949,A -85,B 0,C 180,E1 -445.362,E2 -445.362} C_VEL
LIN {X 0,Y 608.449,Z 400.896,A -85,B 0,C 180,E1 -446.357,E2 -446.357} C_VEL
LIN {X 0,Y 608.425,Z 403.809,A -85,B 0,C 180,E1 -447.352,E2 -447.352} C_VEL
LIN {X 0,Y 608.445,Z 405.201,A -85,B 0,C 180,E1 -448.014,E2 -448.014} C_VEL
LIN {X 0,Y 608.438,Z 406.783,A -85,B 0,C 180,E1 -449.338,E2 -449.338} C_VEL
LIN {X 0,Y 608.434,Z 407,A -85,B 0,C 180,E1 -450,E2 -450} C_VEL
LIN {X 0,Y 608.448,Z 406.184,A -85,B 0,C 180,E1 -451.324,E2 -451.324} C_VEL
LIN {X 0,Y 608.445,Z 405.202,A -85,B 0,C 180,E1 -451.986,E2 -451.986} C_VEL
LIN {X 0,Y 608.425,Z 403.809,A -85,B 0,C 180,E1 -452.648,E2 -452.648} C_VEL
LIN {X 0,Y 608.449,Z 400.897,A -85,B 0,C 180,E1 -453.642,E2 -453.642} C_VEL
LIN {X 0,Y 608.432,Z 396.95,A -85,B 0,C 180,E1 -454.638,E2 -454.638} C_VEL
LIN {X 0,Y 608.438,Z 390.877,A -85,B 0,C 180,E1 -455.801,E2 -455.801} C_VEL
LIN {X 0,Y 608.462,Z 384.236,A -85,B 0,C 180,E1 -456.799,E2 -456.799} C_VEL
LIN {X 0,Y 608.456,Z 375.99,A -85,B 0,C 180,E1 -457.8,E2 -457.8} C_VEL
LIN {X 0,Y 608.472,Z 367.538,A -85,B 0,C 180,E1 -458.636,E2 -458.636} C_VEL
LIN {X 0,Y 608.479,Z 357.093,A -85,B 0,C 180,E1 -459.473,E2 -459.473} C_VEL
LIN {X 0,Y 608.489,Z 346.758,A -85,B 0,C 180,E1 -460.145,E2 -460.145} C_VEL
LIN {X 0,Y 608.519,Z 335.269,A -85,B 0,C 180,E1 -460.74,E2 -460.74} C_VEL
LIN {X 0,Y 608.528,Z 322.893,A -85,B 0,C 180,E1 -461.225,E2 -461.225} C_VEL
LIN {X 0,Y 608.544,Z 309.443,A -85,B 0,C 180,E1 -461.597,E2 -461.597} C_VEL
LIN {X 0,Y 608.553,Z 297.093,A -85,B 0,C 180,E1 -461.808,E2 -461.808} C_VEL
LIN {X 0,Y 608.438,Z 194.439,A -85,B 0,C 180,E1 -463.038,E2 -463.038} C_VEL
LIN {X 0,Y 608.51,Z 172.002,A -85,B 0,C 180,E1 -465.92,E2 -465.92} C_VEL
LIN {X 0,Y 608.5,Z 152.262,A -85,B 0,C 180,E1 -468.492,E2 -468.492} C_VEL
LIN {X 0,Y 608.566,Z 132.114,A -85,B 0,C 180,E1 -471.155,E2 -471.155} C_VEL
LIN {X 0,Y 608.466,Z 117.738,A -85,B 0,C 180,E1 -473.089,E2 -473.089} C_VEL
LIN {X 0,Y 608.475,Z 117.688,A -85,B 0,C 180,E1 -475.721,E2 -475.721} C_VEL
LIN {X 0,Y 608.457,Z 117.689,A -85,B 0,C 180,E1 -478.617,E2 -478.617} C_VEL
LIN {X 0,Y 608.447,Z 117.689,A -85,B 0,C 180,E1 -481.318,E2 -481.318} C_VEL
LIN {X 0,Y 608.476,Z 117.691,A -85,B 0,C 180,E1 -483.735,E2 -483.735} C_VEL
LIN {X 0,Y 608.446,Z 117.696,A -85,B 0,C 180,E1 -486.092,E2 -486.092} C_VEL
LIN {X 0,Y 608.435,Z 117.69,A -85,B 0,C 180,E1 -488.59,E2 -488.59} C_VEL
LIN {X 0,Y 608.464,Z 117.689,A -85,B 0,C 180,E1 -491.342,E2 -491.342} C_VEL
LIN {X 0,Y 608.464,Z 117.694,A -85,B 0,C 180,E1 -493.87,E2 -493.87} C_VEL
LIN {X 0,Y 608.469,Z 117.685,A -85,B 0,C 180,E1 -496.691,E2 -496.691} C_VEL
LIN {X 0,Y 608.453,Z 117.696,A -85,B 0,C 180,E1 -499.696,E2 -499.696} C_VEL
LIN {X 0,Y 608.459,Z 117.688,A -85,B 0,C 180,E1 -502.253,E2 -502.253} C_VEL
LIN {X 0,Y 608.452,Z 117.692,A -85,B 0,C 180,E1 -505.094,E2 -505.094} C_VEL
LIN {X 0,Y 608.455,Z 117.69,A -85,B 0,C 180,E1 -507.905,E2 -507.905} C_VEL
LIN {X 0,Y 608.452,Z 117.688,A -85,B 0,C 180,E1 -510.219,E2 -510.219} C_VEL
LIN {X 0,Y 608.482,Z 117.686,A -85,B 0,C 180,E1 -512.792,E2 -512.792} C_VEL
LIN {X 0,Y 608.444,Z 117.696,A -85,B 0,C 180,E1 -515.428,E2 -515.428} C_VEL
LIN {X 0,Y 608.465,Z 117.686,A -85,B 0,C 180,E1 -518.308,E2 -518.308} C_VEL
LIN {X 0,Y 608.465,Z 117.693,A -85,B 0,C 180,E1 -521.285,E2 -521.285} C_VEL
LIN {X 0,Y 608.447,Z 117.688,A -85,B 0,C 180,E1 -523.906,E2 -523.906} C_VEL
LIN {X 0,Y 608.466,Z 117.691,A -85,B 0,C 180,E1 -526.643,E2 -526.643} C_VEL
LIN {X 0,Y 608.448,Z 117.692,A -85,B 0,C 180,E1 -529.35,E2 -529.35} C_VEL
LIN {X 0,Y 608.474,Z 117.685,A -85,B 0,C 180,E1 -532.033,E2 -532.033} C_VEL
LIN {X 0,Y 608.472,Z 117.694,A -85,B 0,C 180,E1 -534.698,E2 -534.698} C_VEL
LIN {X 0,Y 608.456,Z 117.689,A -85,B 0,C 180,E1 -537.352,E2 -537.352} C_VEL
LIN {X 0,Y 608.477,Z 117.685,A -85,B 0,C 180,E1 -540,E2 -540} C_VEL
LIN {X 0,Y 608.481,Z 117.695,A -85,B 0,C 180,E1 -542.648,E2 -542.648} C_VEL
LIN {X 0,Y 608.442,Z 117.69,A -85,B 0,C 180,E1 -545.302,E2 -545.302} C_VEL
LIN {X 0,Y 608.479,Z 117.687,A -85,B 0,C 180,E1 -547.967,E2 -547.967} C_VEL
LIN {X 0,Y 608.448,Z 117.688,A -85,B 0,C 180,E1 -549.461,E2 -549.461} C_VEL
LIN {X 0,Y 607.784,Z 117.775,A -85,B 0,C 180,E1 -550.013,E2 -550.013} C_VEL
LIN {X 0,Y 604.936,Z 118.13,A -85,B 0,C 180,E1 -550.91,E2 -550.91} C_VEL
LIN {X 0,Y 602.528,Z 118.431,A -85,B 0,C 180,E1 -551.631,E2 -551.631} C_VEL
LIN {X 0,Y 601.491,Z 118.561,A -85,B 0,C 180,E1 -552.188,E2 -552.188} C_VEL
LIN {X 0,Y 601.405,Z 118.569,A -85,B 0,C 180,E1 -552.376,E2 -552.376} C_VEL
LIN {X 0,Y 601.422,Z 118.565,A -85,B 0,C 180,E1 -554.897,E2 -554.897} C_VEL
LIN {X 0,Y 601.409,Z 118.566,A -85,B 0,C 180,E1 -556.986,E2 -556.986} C_VEL
LIN {X 0,Y 601.403,Z 118.569,A -85,B 0,C 180,E1 -559.809,E2 -559.809} C_VEL
LIN {X 0,Y 601.41,Z 118.567,A -85,B 0,C 180,E1 -562.683,E2 -562.683} C_VEL
LIN {X 0,Y 601.395,Z 118.567,A -85,B 0,C 180,E1 -564.879,E2 -564.879} C_VEL
LIN {X 0,Y 601.411,Z 118.566,A -85,B 0,C 180,E1 -567.362,E2 -567.362} C_VEL
LIN {X 0,Y 601.428,Z 118.57,A -85,B 0,C 180,E1 -570.164,E2 -570.164} C_VEL
LIN {X 0,Y 601.409,Z 118.565,A -85,B 0,C 180,E1 -572.714,E2 -572.714} C_VEL
LIN {X 0,Y 601.388,Z 118.568,A -85,B 0,C 180,E1 -575.111,E2 -575.111} C_VEL
LIN {X 0,Y 601.435,Z 118.565,A -85,B 0,C 180,E1 -577.419,E2 -577.419} C_VEL
LIN {X 0,Y 601.412,Z 118.571,A -85,B 0,C 180,E1 -579.995,E2 -579.995} C_VEL
LIN {X 0,Y 601.404,Z 118.565,A -85,B 0,C 180,E1 -582.671,E2 -582.671} C_VEL
LIN {X 0,Y 601.426,Z 118.57,A -85,B 0,C 180,E1 -585.482,E2 -585.482} C_VEL
LIN {X 0,Y 601.417,Z 118.564,A -85,B 0,C 180,E1 -588.408,E2 -588.408} C_VEL
LIN {X 0,Y 601.413,Z 118.566,A -85,B 0,C 180,E1 -590.874,E2 -590.874} C_VEL
LIN {X 0,Y 601.404,Z 118.575,A -85,B 0,C 180,E1 -593.417,E2 -593.417} C_VEL
LIN {X 0,Y 601.416,Z 118.565,A -85,B 0,C 180,E1 -596.067,E2 -596.067} C_VEL
LIN {X 0,Y 601.418,Z 118.564,A -85,B 0,C 180,E1 -598.546,E2 -598.546} C_VEL
LIN {X 0,Y 601.429,Z 118.572,A -85,B 0,C 180,E1 -601.373,E2 -601.373} C_VEL
LIN {X 0,Y 601.395,Z 118.571,A -85,B 0,C 180,E1 -603.636,E2 -603.636} C_VEL
LIN {X 0,Y 601.437,Z 118.563,A -85,B 0,C 180,E1 -605.859,E2 -605.859} C_VEL
LIN {X 0,Y 601.407,Z 118.57,A -85,B 0,C 180,E1 -608.761,E2 -608.761} C_VEL
LIN {X 0,Y 601.392,Z 118.569,A -85,B 0,C 180,E1 -611.607,E2 -611.607} C_VEL
LIN {X 0,Y 601.411,Z 118.566,A -85,B 0,C 180,E1 -614.409,E2 -614.409} C_VEL
LIN {X 0,Y 601.409,Z 118.571,A -85,B 0,C 180,E1 -617.172,E2 -617.172} C_VEL
LIN {X 0,Y 601.43,Z 118.562,A -85,B 0,C 180,E1 -619.905,E2 -619.905} C_VEL
LIN {X 0,Y 601.442,Z 118.568,A -85,B 0,C 180,E1 -622.615,E2 -622.615} C_VEL
LIN {X 0,Y 601.403,Z 118.568,A -85,B 0,C 180,E1 -625.308,E2 -625.308} C_VEL
LIN {X 0,Y 601.436,Z 118.563,A -85,B 0,C 180,E1 -627.991,E2 -627.991} C_VEL
LIN {X 0,Y 601.451,Z 118.57,A -85,B 0,C 180,E1 -630.67,E2 -630.67} C_VEL
LIN {X 0,Y 601.443,Z 118.717,A -85,B 0,C 180,E1 -631.925,E2 -631.925} C_VEL
LIN {X 0,Y 601.398,Z 134.208,A -85,B 0,C 180,E1 -634.692,E2 -634.692} C_VEL
LIN {X 0,Y 601.378,Z 146.603,A -85,B 0,C 180,E1 -636.88,E2 -636.88} C_VEL
LIN {X 0,Y 601.643,Z 152.958,A -85,B 0,C 180,E1 -636.972,E2 -636.972} C_VEL
LIN {X 0,Y 601.546,Z 253.11,A -85,B 0,C 180,E1 -638.186,E2 -638.186} C_VEL
LIN {X 0,Y 601.548,Z 266.21,A -85,B 0,C 180,E1 -638.482,E2 -638.482} C_VEL
LIN {X 0,Y 601.528,Z 278.844,A -85,B 0,C 180,E1 -638.906,E2 -638.906} C_VEL
LIN {X 0,Y 601.537,Z 290.109,A -85,B 0,C 180,E1 -639.414,E2 -639.414} C_VEL
LIN {X 0,Y 601.466,Z 301.81,A -85,B 0,C 180,E1 -640.095,E2 -640.095} C_VEL
LIN {X 0,Y 601.436,Z 312.476,A -85,B 0,C 180,E1 -640.874,E2 -640.874} C_VEL
LIN {X 0,Y 601.433,Z 320.936,A -85,B 0,C 180,E1 -641.629,E2 -641.629} C_VEL
LIN {X 0,Y 601.398,Z 328.919,A -85,B 0,C 180,E1 -642.486,E2 -642.486} C_VEL
LIN {X 0,Y 601.372,Z 336.717,A -85,B 0,C 180,E1 -643.517,E2 -643.517} C_VEL
LIN {X 0,Y 601.34,Z 342.996,A -85,B 0,C 180,E1 -644.553,E2 -644.553} C_VEL
LIN {X 0,Y 601.339,Z 347.97,A -85,B 0,C 180,E1 -645.593,E2 -645.593} C_VEL
LIN {X 0,Y 601.327,Z 351.626,A -85,B 0,C 180,E1 -646.59,E2 -646.59} C_VEL
LIN {X 0,Y 601.314,Z 354.52,A -85,B 0,C 180,E1 -647.691,E2 -647.691} C_VEL
LIN {X 0,Y 601.343,Z 356.292,A -85,B 0,C 180,E1 -648.798,E2 -648.798} C_VEL
LIN {X 0,Y 601.316,Z 356.952,A -85,B 0,C 180,E1 -649.813,E2 -649.813} C_VEL
LIN {X 0,Y 601.341,Z 356.741,A -85,B 0,C 180,E1 -650.776,E2 -650.776} C_VEL
LIN {X 0,Y 601.339,Z 355.353,A -85,B 0,C 180,E1 -651.962,E2 -651.962} C_VEL
LIN {X 0,Y 601.355,Z 352.955,A -85,B 0,C 180,E1 -653.049,E2 -653.049} C_VEL
LIN {X 0,Y 601.328,Z 348.921,A -85,B 0,C 180,E1 -654.27,E2 -654.27} C_VEL
LIN {X 0,Y 601.374,Z 344.519,A -85,B 0,C 180,E1 -655.25,E2 -655.25} C_VEL
LIN {X 0,Y 601.385,Z 338.101,A -85,B 0,C 180,E1 -656.365,E2 -656.365} C_VEL
LIN {X 0,Y 601.398,Z 330.907,A -85,B 0,C 180,E1 -657.359,E2 -657.359} C_VEL
LIN {X 0,Y 601.414,Z 323.057,A -85,B 0,C 180,E1 -658.247,E2 -658.247} C_VEL
LIN {X 0,Y 601.462,Z 313.726,A -85,B 0,C 180,E1 -659.114,E2 -659.114} C_VEL
LIN {X 0,Y 601.447,Z 303.653,A -85,B 0,C 180,E1 -659.873,E2 -659.873} C_VEL
LIN {X 0,Y 601.476,Z 292.488,A -85,B 0,C 180,E1 -660.549,E2 -660.549} C_VEL
LIN {X 0,Y 601.548,Z 280.853,A -85,B 0,C 180,E1 -661.103,E2 -661.103} C_VEL
LIN {X 0,Y 601.579,Z 268.52,A -85,B 0,C 180,E1 -661.542,E2 -661.542} C_VEL
LIN {X 0,Y 601.582,Z 255.188,A -85,B 0,C 180,E1 -661.864,E2 -661.864} C_VEL
LIN {X 0,Y 601.613,Z 234.138,A -85,B 0,C 180,E1 -662.146,E2 -662.146} C_VEL
LIN {X 0,Y 601.608,Z 147.96,A -85,B 0,C 180,E1 -663.179,E2 -663.179} C_VEL
LIN {X 0,Y 601.418,Z 146.571,A -85,B 0,C 180,E1 -663.214,E2 -663.214} C_VEL
LIN {X 0,Y 601.443,Z 130.768,A -85,B 0,C 180,E1 -666.008,E2 -666.008} C_VEL
LIN {X 0,Y 601.379,Z 118.571,A -85,B 0,C 180,E1 -668.205,E2 -668.205} C_VEL
LIN {X 0,Y 601.412,Z 118.568,A -85,B 0,C 180,E1 -670.875,E2 -670.875} C_VEL
LIN {X 0,Y 601.406,Z 118.572,A -85,B 0,C 180,E1 -673.588,E2 -673.588} C_VEL
LIN {X 0,Y 601.404,Z 118.567,A -85,B 0,C 180,E1 -676.43,E2 -676.43} C_VEL
LIN {X 0,Y 601.404,Z 118.571,A -85,B 0,C 180,E1 -679.428,E2 -679.428} C_VEL
LIN {X 0,Y 601.382,Z 118.57,A -85,B 0,C 180,E1 -681.729,E2 -681.729} C_VEL
LIN {X 0,Y 601.368,Z 118.571,A -85,B 0,C 180,E1 -684.244,E2 -684.244} C_VEL
LIN {X 0,Y 601.409,Z 118.572,A -85,B 0,C 180,E1 -686.685,E2 -686.685} C_VEL
LIN {X 0,Y 601.392,Z 118.574,A -85,B 0,C 180,E1 -689.057,E2 -689.057} C_VEL
LIN {X 0,Y 601.387,Z 118.57,A -85,B 0,C 180,E1 -691.371,E2 -691.371} C_VEL
LIN {X 0,Y 601.369,Z 118.57,A -85,B 0,C 180,E1 -693.635,E2 -693.635} C_VEL
LIN {X 0,Y 601.39,Z 118.568,A -85,B 0,C 180,E1 -695.857,E2 -695.857} C_VEL
LIN {X 0,Y 601.389,Z 118.574,A -85,B 0,C 180,E1 -698.76,E2 -698.76} C_VEL
LIN {X 0,Y 601.353,Z 118.572,A -85,B 0,C 180,E1 -701.606,E2 -701.606} C_VEL
LIN {X 0,Y 601.379,Z 118.578,A -85,B 0,C 180,E1 -704.408,E2 -704.408} C_VEL
LIN {X 0,Y 601.345,Z 118.573,A -85,B 0,C 180,E1 -707.17,E2 -707.17} C_VEL
LIN {X 0,Y 601.417,Z 118.569,A -85,B 0,C 180,E1 -709.905,E2 -709.905} C_VEL
LIN {X 0,Y 601.367,Z 118.573,A -85,B 0,C 180,E1 -712.614,E2 -712.614} C_VEL
LIN {X 0,Y 601.386,Z 118.57,A -85,B 0,C 180,E1 -714.636,E2 -714.636} C_VEL
LIN {X 0,Y 601.396,Z 118.568,A -85,B 0,C 180,E1 -717.321,E2 -717.321} C_VEL
LIN {X 0,Y 601.443,Z 118.569,A -85,B 0,C 180,E1 -720,E2 -720} C_VEL
LIN {X 0,Y 601.394,Z 118.567,A -85,B 0,C 180,E1 -722.679,E2 -722.679} C_VEL
LIN {X 0,Y 601.399,Z 118.571,A -85,B 0,C 180,E1 -725.364,E2 -725.364} C_VEL
LIN {X 0,Y 601.428,Z 118.566,A -85,B 0,C 180,E1 -728.061,E2 -728.061} C_VEL
LIN {X 0,Y 601.397,Z 118.569,A -85,B 0,C 180,E1 -730.997,E2 -730.997} C_VEL
LIN {X 0,Y 601.398,Z 118.576,A -85,B 0,C 180,E1 -733.516,E2 -733.516} C_VEL
LIN {X 0,Y 601.394,Z 118.567,A -85,B 0,C 180,E1 -736.288,E2 -736.288} C_VEL
LIN {X 0,Y 601.409,Z 118.572,A -85,B 0,C 180,E1 -739.099,E2 -739.099} C_VEL
LIN {X 0,Y 601.394,Z 118.567,A -85,B 0,C 180,E1 -741.96,E2 -741.96} C_VEL
LIN {X 0,Y 601.391,Z 118.574,A -85,B 0,C 180,E1 -744.879,E2 -744.879} C_VEL
LIN {X 0,Y 601.417,Z 118.569,A -85,B 0,C 180,E1 -747.362,E2 -747.362} C_VEL
LIN {X 0,Y 601.4,Z 118.567,A -85,B 0,C 180,E1 -750.166,E2 -750.166} C_VEL
LIN {X 0,Y 601.407,Z 118.573,A -85,B 0,C 180,E1 -752.713,E2 -752.713} C_VEL
LIN {X 0,Y 601.398,Z 118.571,A -85,B 0,C 180,E1 -755.112,E2 -755.112} C_VEL
LIN {X 0,Y 601.434,Z 118.563,A -85,B 0,C 180,E1 -757.419,E2 -757.419} C_VEL
LIN {X 0,Y 601.4,Z 118.568,A -85,B 0,C 180,E1 -759.996,E2 -759.996} C_VEL
LIN {X 0,Y 601.411,Z 118.573,A -85,B 0,C 180,E1 -762.671,E2 -762.671} C_VEL
LIN {X 0,Y 601.401,Z 118.566,A -85,B 0,C 180,E1 -765.479,E2 -765.479} C_VEL
LIN {X 0,Y 601.422,Z 118.574,A -85,B 0,C 180,E1 -768.407,E2 -768.407} C_VEL
LIN {X 0,Y 601.431,Z 118.564,A -85,B 0,C 180,E1 -770.875,E2 -770.875} C_VEL
LIN {X 0,Y 601.397,Z 118.567,A -85,B 0,C 180,E1 -773.416,E2 -773.416} C_VEL
LIN {X 0,Y 601.432,Z 118.571,A -85,B 0,C 180,E1 -776.065,E2 -776.065} C_VEL
LIN {X 0,Y 601.404,Z 118.566,A -85,B 0,C 180,E1 -779.057,E2 -779.057} C_VEL
LIN {X 0,Y 601.414,Z 118.567,A -85,B 0,C 180,E1 -781.372,E2 -781.372} C_VEL
LIN {X 0,Y 601.395,Z 118.573,A -85,B 0,C 180,E1 -783.636,E2 -783.636} C_VEL
LIN {X 0,Y 601.421,Z 118.568,A -85,B 0,C 180,E1 -786.59,E2 -786.59} C_VEL
LIN {X 0,Y 601.449,Z 118.816,A -85,B 0,C 180,E1 -786.773,E2 -786.773} C_VEL
LIN {X 0,Y 601.695,Z 125.509,A -85,B 0,C 180,E1 -787.696,E2 -787.696} C_VEL
LIN {X 0,Y 601.617,Z 146.738,A -85,B 0,C 180,E1 -790.553,E2 -790.553} C_VEL
LIN {X 0,Y 601.512,Z 167.904,A -85,B 0,C 180,E1 -793.352,E2 -793.352} C_VEL
LIN {X 0,Y 601.467,Z 189.67,A -85,B 0,C 180,E1 -796.19,E2 -796.19} C_VEL
LIN {X 0,Y 601.425,Z 194.521,A -85,B 0,C 180,E1 -796.818,E2 -796.818} C_VEL
LIN {X 0,Y 601.638,Z 207.652,A -85,B 0,C 180,E1 -796.983,E2 -796.983} C_VEL
LIN {X 0,Y 601.613,Z 302.939,A -85,B 0,C 180,E1 -798.139,E2 -798.139} C_VEL
LIN {X 0,Y 601.56,Z 316.213,A -85,B 0,C 180,E1 -798.437,E2 -798.437} C_VEL
LIN {X 0,Y 601.543,Z 328.633,A -85,B 0,C 180,E1 -798.853,E2 -798.853} C_VEL
LIN {X 0,Y 601.523,Z 340.63,A -85,B 0,C 180,E1 -799.396,E2 -799.396} C_VEL
LIN {X 0,Y 601.483,Z 352.197,A -85,B 0,C 180,E1 -800.076,E2 -800.076} C_VEL
LIN {X 0,Y 601.444,Z 362.594,A -85,B 0,C 180,E1 -800.839,E2 -800.839} C_VEL
LIN {X 0,Y 601.429,Z 371.111,A -85,B 0,C 180,E1 -801.601,E2 -801.601} C_VEL
LIN {X 0,Y 601.418,Z 378.959,A -85,B 0,C 180,E1 -802.446,E2 -802.446} C_VEL
LIN {X 0,Y 601.37,Z 386.224,A -85,B 0,C 180,E1 -803.398,E2 -803.398} C_VEL
LIN {X 0,Y 601.372,Z 391.865,A -85,B 0,C 180,E1 -804.299,E2 -804.299} C_VEL
LIN {X 0,Y 601.336,Z 396.949,A -85,B 0,C 180,E1 -805.307,E2 -805.307} C_VEL
LIN {X 0,Y 601.368,Z 400.896,A -85,B 0,C 180,E1 -806.315,E2 -806.315} C_VEL
LIN {X 0,Y 601.325,Z 403.809,A -85,B 0,C 180,E1 -807.32,E2 -807.32} C_VEL
LIN {X 0,Y 601.343,Z 405.201,A -85,B 0,C 180,E1 -807.991,E2 -807.991} C_VEL
LIN {X 0,Y 601.339,Z 406.784,A -85,B 0,C 180,E1 -809.33,E2 -809.33} C_VEL
LIN {X 0,Y 601.335,Z 407,A -85,B 0,C 180,E1 -810,E2 -810} C_VEL
LIN {X 0,Y 601.347,Z 406.185,A -85,B 0,C 180,E1 -811.339,E2 -811.339} C_VEL
LIN {X 0,Y 601.344,Z 405.202,A -85,B 0,C 180,E1 -812.009,E2 -812.009} C_VEL
LIN {X 0,Y 601.325,Z 403.81,A -85,B 0,C 180,E1 -812.679,E2 -812.679} C_VEL
LIN {X 0,Y 601.368,Z 400.896,A -85,B 0,C 180,E1 -813.685,E2 -813.685} C_VEL
LIN {X 0,Y 601.336,Z 396.95,A -85,B 0,C 180,E1 -814.693,E2 -814.693} C_VEL
LIN {X 0,Y 601.373,Z 390.878,A -85,B 0,C 180,E1 -815.869,E2 -815.869} C_VEL
LIN {X 0,Y 601.382,Z 384.237,A -85,B 0,C 180,E1 -816.88,E2 -816.88} C_VEL
LIN {X 0,Y 601.4,Z 375.991,A -85,B 0,C 180,E1 -817.892,E2 -817.892} C_VEL
LIN {X 0,Y 601.436,Z 367.538,A -85,B 0,C 180,E1 -818.737,E2 -818.737} C_VEL
LIN {X 0,Y 601.449,Z 357.095,A -85,B 0,C 180,E1 -819.585,E2 -819.585} C_VEL
LIN {X 0,Y 601.467,Z 346.76,A -85,B 0,C 180,E1 -820.264,E2 -820.264} C_VEL
LIN {X 0,Y 601.538,Z 334.599,A -85,B 0,C 180,E1 -820.896,E2 -820.896} C_VEL
LIN {X 0,Y 601.555,Z 322.221,A -85,B 0,C 180,E1 -821.379,E2 -821.379} C_VEL
LIN {X 0,Y 601.583,Z 309.442,A -85,B 0,C 180,E1 -821.733,E2 -821.733} C_VEL
LIN {X 0,Y 601.623,Z 297.093,A -85,B 0,C 180,E1 -821.946,E2 -821.946} C_VEL
LIN {X 0,Y 601.505,Z 195.152,A -85,B 0,C 180,E1 -823.17,E2 -823.17} C_VEL
LIN {X 0,Y 601.444,Z 194.273,A -85,B 0,C 180,E1 -823.214,E2 -823.214} C_VEL
LIN {X 0,Y 601.516,Z 172.002,A -85,B 0,C 180,E1 -826.11,E2 -826.11} C_VEL
LIN {X 0,Y 601.532,Z 152.092,A -85,B 0,C 180,E1 -828.737,E2 -828.737} C_VEL
LIN {X 0,Y 601.656,Z 132.114,A -85,B 0,C 180,E1 -831.41,E2 -831.41} C_VEL
LIN {X 0,Y 601.673,Z 120.148,A -85,B 0,C 180,E1 -833.036,E2 -833.036} C_VEL
LIN {X 0,Y 601.409,Z 118.569,A -85,B 0,C 180,E1 -833.274,E2 -833.274} C_VEL
LIN {X 0,Y 601.413,Z 118.571,A -85,B 0,C 180,E1 -835.867,E2 -835.867} C_VEL
LIN {X 0,Y 601.401,Z 118.573,A -85,B 0,C 180,E1 -837.868,E2 -837.868} C_VEL
LIN {X 0,Y 601.43,Z 118.571,A -85,B 0,C 180,E1 -840.164,E2 -840.164} C_VEL
LIN {X 0,Y 601.412,Z 118.565,A -85,B 0,C 180,E1 -842.713,E2 -842.713} C_VEL
LIN {X 0,Y 601.389,Z 118.568,A -85,B 0,C 180,E1 -845.111,E2 -845.111} C_VEL
LIN {X 0,Y 601.437,Z 118.565,A -85,B 0,C 180,E1 -847.419,E2 -847.419} C_VEL
LIN {X 0,Y 601.413,Z 118.572,A -85,B 0,C 180,E1 -849.995,E2 -849.995} C_VEL
LIN {X 0,Y 601.407,Z 118.565,A -85,B 0,C 180,E1 -852.671,E2 -852.671} C_VEL
LIN {X 0,Y 601.428,Z 118.569,A -85,B 0,C 180,E1 -855.482,E2 -855.482} C_VEL
LIN {X 0,Y 601.418,Z 118.564,A -85,B 0,C 180,E1 -858.407,E2 -858.407} C_VEL
LIN {X 0,Y 601.414,Z 118.565,A -85,B 0,C 180,E1 -860.873,E2 -860.873} C_VEL
LIN {X 0,Y 601.404,Z 118.574,A -85,B 0,C 180,E1 -863.417,E2 -863.417} C_VEL
LIN {X 0,Y 601.417,Z 118.566,A -85,B 0,C 180,E1 -866.066,E2 -866.066} C_VEL
LIN {X 0,Y 601.419,Z 118.564,A -85,B 0,C 180,E1 -868.545,E2 -868.545} C_VEL
LIN {X 0,Y 601.431,Z 118.572,A -85,B 0,C 180,E1 -871.373,E2 -871.373} C_VEL
LIN {X 0,Y 601.396,Z 118.571,A -85,B 0,C 180,E1 -873.636,E2 -873.636} C_VEL
LIN {X 0,Y 601.416,Z 118.566,A -85,B 0,C 180,E1 -876.589,E2 -876.589} C_VEL
LIN {X 0,Y 601.422,Z 118.568,A -85,B 0,C 180,E1 -879.478,E2 -879.478} C_VEL
LIN {X 0,Y 601.391,Z 118.568,A -85,B 0,C 180,E1 -882.311,E2 -882.311} C_VEL
LIN {X 0,Y 601.423,Z 118.572,A -85,B 0,C 180,E1 -885.103,E2 -885.103} C_VEL
LIN {X 0,Y 601.411,Z 118.565,A -85,B 0,C 180,E1 -887.857,E2 -887.857} C_VEL
LIN {X 0,Y 601.421,Z 118.568,A -85,B 0,C 180,E1 -890.584,E2 -890.584} C_VEL
LIN {X 0,Y 601.401,Z 118.569,A -85,B 0,C 180,E1 -893.289,E2 -893.289} C_VEL
LIN {X 0,Y 601.404,Z 118.566,A -85,B 0,C 180,E1 -895.979,E2 -895.979} C_VEL
LIN {X 0,Y 601.43,Z 118.572,A -85,B 0,C 180,E1 -898.661,E2 -898.661} C_VEL
LIN {X 0,Y 601.403,Z 118.567,A -85,B 0,C 180,E1 -901.339,E2 -901.339} C_VEL
LIN {X 0,Y 601.411,Z 118.565,A -85,B 0,C 180,E1 -903.35,E2 -903.35} C_VEL
LIN {X 0,Y 601.443,Z 118.563,A -85,B 0,C 180,E1 -906.037,E2 -906.037} C_VEL
LIN {X 0,Y 601.411,Z 118.571,A -85,B 0,C 180,E1 -908.738,E2 -908.738} C_VEL
LIN {X 0,Y 601.41,Z 118.565,A -85,B 0,C 180,E1 -911.458,E2 -911.458} C_VEL
LIN {X 0,Y 601.405,Z 118.569,A -85,B 0,C 180,E1 -912.376,E2 -912.376} C_VEL
LIN {X 0,Y 600.736,Z 118.652,A -85,B 0,C 180,E1 -912.936,E2 -912.936} C_VEL
LIN {X 0,Y 597.884,Z 119.006,A -85,B 0,C 180,E1 -913.844,E2 -913.844} C_VEL
LIN {X 0,Y 595.476,Z 119.311,A -85,B 0,C 180,E1 -914.574,E2 -914.574} C_VEL
LIN {X 0,Y 594.44,Z 119.434,A -85,B 0,C 180,E1 -915.138,E2 -915.138} C_VEL
LIN {X 0,Y 594.355,Z 119.444,A -85,B 0,C 180,E1 -915.328,E2 -915.328} C_VEL
LIN {X 0,Y 594.348,Z 119.449,A -85,B 0,C 180,E1 -917.905,E2 -917.905} C_VEL
LIN {X 0,Y 594.394,Z 119.441,A -85,B 0,C 180,E1 -920.776,E2 -920.776} C_VEL
LIN {X 0,Y 594.378,Z 119.444,A -85,B 0,C 180,E1 -923.704,E2 -923.704} C_VEL
LIN {X 0,Y 594.377,Z 119.443,A -85,B 0,C 180,E1 -926.7,E2 -926.7} C_VEL
LIN {X 0,Y 594.374,Z 119.441,A -85,B 0,C 180,E1 -928.999,E2 -928.999} C_VEL
LIN {X 0,Y 594.375,Z 119.446,A -85,B 0,C 180,E1 -931.642,E2 -931.642} C_VEL
LIN {X 0,Y 594.373,Z 119.443,A -85,B 0,C 180,E1 -934.58,E2 -934.58} C_VEL
LIN {X 0,Y 594.388,Z 119.446,A -85,B 0,C 180,E1 -937.608,E2 -937.608} C_VEL
LIN {X 0,Y 594.36,Z 119.443,A -85,B 0,C 180,E1 -940.568,E2 -940.568} C_VEL
LIN {X 0,Y 594.365,Z 119.446,A -85,B 0,C 180,E1 -943.3,E2 -943.3} C_VEL
LIN {X 0,Y 594.366,Z 119.445,A -85,B 0,C 180,E1 -946.161,E2 -946.161} C_VEL
LIN {X 0,Y 594.375,Z 119.441,A -85,B 0,C 180,E1 -948.536,E2 -948.536} C_VEL
LIN {X 0,Y 594.38,Z 119.447,A -85,B 0,C 180,E1 -951.296,E2 -951.296} C_VEL
LIN {X 0,Y 594.348,Z 119.45,A -85,B 0,C 180,E1 -953.755,E2 -953.755} C_VEL
LIN {X 0,Y 594.364,Z 119.443,A -85,B 0,C 180,E1 -956.238,E2 -956.238} C_VEL
LIN {X 0,Y 594.368,Z 119.443,A -85,B 0,C 180,E1 -958.65,E2 -958.65} C_VEL
LIN {X 0,Y 594.382,Z 119.446,A -85,B 0,C 180,E1 -961.042,E2 -961.042} C_VEL
LIN {X 0,Y 594.377,Z 119.442,A -85,B 0,C 180,E1 -963.979,E2 -963.979} C_VEL
LIN {X 0,Y 594.368,Z 119.442,A -85,B 0,C 180,E1 -966.295,E2 -966.295} C_VEL
LIN {X 0,Y 594.398,Z 119.447,A -85,B 0,C 180,E1 -969.224,E2 -969.224} C_VEL
LIN {X 0,Y 594.342,Z 119.445,A -85,B 0,C 180,E1 -972.095,E2 -972.095} C_VEL
LIN {X 0,Y 594.361,Z 119.443,A -85,B 0,C 180,E1 -974.219,E2 -974.219} C_VEL
LIN {X 0,Y 594.38,Z 119.442,A -85,B 0,C 180,E1 -976.321,E2 -976.321} C_VEL
LIN {X 0,Y 594.366,Z 119.449,A -85,B 0,C 180,E1 -979.095,E2 -979.095} C_VEL
LIN {X 0,Y 594.38,Z 119.441,A -85,B 0,C 180,E1 -981.843,E2 -981.843} C_VEL
LIN {X 0,Y 594.403,Z 119.445,A -85,B 0,C 180,E1 -984.572,E2 -984.572} C_VEL
LIN {X 0,Y 594.391,Z 119.441,A -85,B 0,C 180,E1 -987.289,E2 -987.289} C_VEL
LIN {X 0,Y 594.414,Z 119.438,A -85,B 0,C 180,E1 -990,E2 -990} C_VEL
LIN {X 0,Y 594.415,Z 119.594,A -85,B 0,C 180,E1 -991.863,E2 -991.863} C_VEL
LIN {X 0,Y 594.394,Z 133.658,A -85,B 0,C 180,E1 -994.408,E2 -994.408} C_VEL
LIN {X 0,Y 594.34,Z 146.621,A -85,B 0,C 180,E1 -996.725,E2 -996.725} C_VEL
LIN {X 0,Y 594.723,Z 150.452,A -85,B 0,C 180,E1 -996.787,E2 -996.787} C_VEL
LIN {X 0,Y 594.605,Z 253.19,A -85,B 0,C 180,E1 -998.047,E2 -998.047} C_VEL
LIN {X 0,Y 594.583,Z 266.283,A -85,B 0,C 180,E1 -998.347,E2 -998.347} C_VEL
LIN {X 0,Y 594.553,Z 279.454,A -85,B 0,C 180,E1 -998.797,E2 -998.797} C_VEL
LIN {X 0,Y 594.535,Z 291.355,A -85,B 0,C 180,E1 -999.354,E2 -999.354} C_VEL
LIN {X 0,Y 594.437,Z 302.815,A -85,B 0,C 180,E1 -1000.043,E2 -1000.043} C_VEL
LIN {X 0,Y 594.391,Z 313.149,A -85,B 0,C 180,E1 -1000.819,E2 -1000.819} C_VEL
LIN {X 0,Y 594.379,Z 321.631,A -85,B 0,C 180,E1 -1001.596,E2 -1001.596} C_VEL
LIN {X 0,Y 594.346,Z 330.85,A -85,B 0,C 180,E1 -1002.636,E2 -1002.636} C_VEL
LIN {X 0,Y 594.295,Z 338.307,A -85,B 0,C 180,E1 -1003.681,E2 -1003.681} C_VEL
LIN {X 0,Y 594.269,Z 344.282,A -85,B 0,C 180,E1 -1004.73,E2 -1004.73} C_VEL
LIN {X 0,Y 594.271,Z 348.973,A -85,B 0,C 180,E1 -1005.784,E2 -1005.784} C_VEL
LIN {X 0,Y 594.242,Z 352.005,A -85,B 0,C 180,E1 -1006.67,E2 -1006.67} C_VEL
LIN {X 0,Y 594.209,Z 355.03,A -85,B 0,C 180,E1 -1007.91,E2 -1007.91} C_VEL
LIN {X 0,Y 594.242,Z 356.415,A -85,B 0,C 180,E1 -1008.889,E2 -1008.889} C_VEL
LIN {X 0,Y 594.22,Z 357,A -85,B 0,C 180,E1 -1010.059,E2 -1010.059} C_VEL
LIN {X 0,Y 594.25,Z 356.674,A -85,B 0,C 180,E1 -1010.884,E2 -1010.884} C_VEL
LIN {X 0,Y 594.253,Z 354.918,A -85,B 0,C 180,E1 -1012.238,E2 -1012.238} C_VEL
LIN {X 0,Y 594.241,Z 352.25,A -85,B 0,C 180,E1 -1013.341,E2 -1013.341} C_VEL
LIN {X 0,Y 594.25,Z 348.378,A -85,B 0,C 180,E1 -1014.452,E2 -1014.452} C_VEL
LIN {X 0,Y 594.259,Z 343.15,A -85,B 0,C 180,E1 -1015.574,E2 -1015.574} C_VEL
LIN {X 0,Y 594.291,Z 336.369,A -85,B 0,C 180,E1 -1016.704,E2 -1016.704} C_VEL
LIN {X 0,Y 594.344,Z 329.414,A -85,B 0,C 180,E1 -1017.634,E2 -1017.634} C_VEL
LIN {X 0,Y 594.383,Z 320.413,A -85,B 0,C 180,E1 -1018.612,E2 -1018.612} C_VEL
LIN {X 0,Y 594.428,Z 310.543,A -85,B 0,C 180,E1 -1019.481,E2 -1019.481} C_VEL
LIN {X 0,Y 594.453,Z 299.483,A -85,B 0,C 180,E1 -1020.266,E2 -1020.266} C_VEL
LIN {X 0,Y 594.527,Z 287.219,A -85,B 0,C 180,E1 -1020.946,E2 -1020.946} C_VEL
LIN {X 0,Y 594.614,Z 275.225,A -85,B 0,C 180,E1 -1021.454,E2 -1021.454} C_VEL
LIN {X 0,Y 594.631,Z 262.775,A -85,B 0,C 180,E1 -1021.838,E2 -1021.838} C_VEL
LIN {X 0,Y 594.662,Z 249.878,A -85,B 0,C 180,E1 -1022.093,E2 -1022.093} C_VEL
LIN {X 0,Y 594.655,Z 148.376,A -85,B 0,C 180,E1 -1023.33,E2 -1023.33} C_VEL
LIN {X 0,Y 594.375,Z 146.532,A -85,B 0,C 180,E1 -1023.38,E2 -1023.38} C_VEL
LIN {X 0,Y 594.406,Z 130.552,A -85,B 0,C 180,E1 -1026.241,E2 -1026.241} C_VEL
LIN {X 0,Y 594.358,Z 119.447,A -85,B 0,C 180,E1 -1028.266,E2 -1028.266} C_VEL
LIN {X 0,Y 594.373,Z 119.444,A -85,B 0,C 180,E1 -1030.822,E2 -1030.822} C_VEL
LIN {X 0,Y 594.344,Z 119.448,A -85,B 0,C 180,E1 -1033.837,E2 -1033.837} C_VEL
LIN {X 0,Y 594.344,Z 119.448,A -85,B 0,C 180,E1 -1036.699,E2 -1036.699} C_VEL
LIN {X 0,Y 594.358,Z 119.449,A -85,B 0,C 180,E1 -1039.432,E2 -1039.432} C_VEL
LIN {X 0,Y 594.381,Z 119.442,A -85,B 0,C 180,E1 -1042.393,E2 -1042.393} C_VEL
LIN {X 0,Y 594.361,Z 119.446,A -85,B 0,C 180,E1 -1045.419,E2 -1045.419} C_VEL
LIN {X 0,Y 594.338,Z 119.446,A -85,B 0,C 180,E1 -1047.851,E2 -1047.851} C_VEL
LIN {X 0,Y 594.333,Z 119.449,A -85,B 0,C 180,E1 -1050.221,E2 -1050.221} C_VEL
LIN {X 0,Y 594.355,Z 119.446,A -85,B 0,C 180,E1 -1053.299,E2 -1053.299} C_VEL
LIN {X 0,Y 594.331,Z 119.447,A -85,B 0,C 180,E1 -1055.579,E2 -1055.579} C_VEL
LIN {X 0,Y 594.343,Z 119.455,A -85,B 0,C 180,E1 -1058.496,E2 -1058.496} C_VEL
LIN {X 0,Y 594.327,Z 119.447,A -85,B 0,C 180,E1 -1061.381,E2 -1061.381} C_VEL
LIN {X 0,Y 594.326,Z 119.455,A -85,B 0,C 180,E1 -1064.218,E2 -1064.218} C_VEL
LIN {X 0,Y 594.301,Z 119.451,A -85,B 0,C 180,E1 -1067.016,E2 -1067.016} C_VEL
LIN {X 0,Y 594.316,Z 119.448,A -85,B 0,C 180,E1 -1069.094,E2 -1069.094} C_VEL
LIN {X 0,Y 594.351,Z 119.45,A -85,B 0,C 180,E1 -1071.843,E2 -1071.843} C_VEL
LIN {X 0,Y 594.356,Z 119.446,A -85,B 0,C 180,E1 -1074.572,E2 -1074.572} C_VEL
LIN {X 0,Y 594.364,Z 119.444,A -85,B 0,C 180,E1 -1077.289,E2 -1077.289} C_VEL
LIN {X 0,Y 594.412,Z 119.445,A -85,B 0,C 180,E1 -1080,E2 -1080} C_VEL
LIN {X 0,Y 594.363,Z 119.442,A -85,B 0,C 180,E1 -1082.711,E2 -1082.711} C_VEL
LIN {X 0,Y 594.367,Z 119.448,A -85,B 0,C 180,E1 -1085.428,E2 -1085.428} C_VEL
LIN {X 0,Y 594.371,Z 119.444,A -85,B 0,C 180,E1 -1088.157,E2 -1088.157} C_VEL
LIN {X 0,Y 594.366,Z 119.446,A -85,B 0,C 180,E1 -1091.061,E2 -1091.061} C_VEL
LIN {X 0,Y 594.356,Z 119.444,A -85,B 0,C 180,E1 -1094.16,E2 -1094.16} C_VEL
LIN {X 0,Y 594.37,Z 119.45,A -85,B 0,C 180,E1 -1097.194,E2 -1097.194} C_VEL
LIN {X 0,Y 594.354,Z 119.444,A -85,B 0,C 180,E1 -1100.055,E2 -1100.055} C_VEL
LIN {X 0,Y 594.349,Z 119.451,A -85,B 0,C 180,E1 -1102.968,E2 -1102.968} C_VEL
LIN {X 0,Y 594.368,Z 119.442,A -85,B 0,C 180,E1 -1106.019,E2 -1106.019} C_VEL
LIN {X 0,Y 594.33,Z 119.448,A -85,B 0,C 180,E1 -1108.23,E2 -1108.23} C_VEL
LIN {X 0,Y 594.366,Z 119.446,A -85,B 0,C 180,E1 -1110.561,E2 -1110.561} C_VEL
LIN {X 0,Y 594.375,Z 119.45,A -85,B 0,C 180,E1 -1112.951,E2 -1112.951} C_VEL
LIN {X 0,Y 594.35,Z 119.446,A -85,B 0,C 180,E1 -1115.409,E2 -1115.409} C_VEL
LIN {X 0,Y 594.373,Z 119.442,A -85,B 0,C 180,E1 -1117.942,E2 -1117.942} C_VEL
LIN {X 0,Y 594.372,Z 119.449,A -85,B 0,C 180,E1 -1120.821,E2 -1120.821} C_VEL
LIN {X 0,Y 594.353,Z 119.445,A -85,B 0,C 180,E1 -1123.301,E2 -1123.301} C_VEL
LIN {X 0,Y 594.362,Z 119.449,A -85,B 0,C 180,E1 -1126.161,E2 -1126.161} C_VEL
LIN {X 0,Y 594.375,Z 119.442,A -85,B 0,C 180,E1 -1129.179,E2 -1129.179} C_VEL
LIN {X 0,Y 594.38,Z 119.448,A -85,B 0,C 180,E1 -1132.059,E2 -1132.059} C_VEL
LIN {X 0,Y 594.351,Z 119.447,A -85,B 0,C 180,E1 -1134.677,E2 -1134.677} C_VEL
LIN {X 0,Y 594.377,Z 119.442,A -85,B 0,C 180,E1 -1137.089,E2 -1137.089} C_VEL
LIN {X 0,Y 594.373,Z 119.447,A -85,B 0,C 180,E1 -1139.675,E2 -1139.675} C_VEL
LIN {X 0,Y 594.378,Z 119.443,A -85,B 0,C 180,E1 -1142.539,E2 -1142.539} C_VEL
LIN {X 0,Y 594.374,Z 119.443,A -85,B 0,C 180,E1 -1144.807,E2 -1144.807} C_VEL
LIN {X 0,Y 594.39,Z 119.459,A -85,B 0,C 180,E1 -1146.573,E2 -1146.573} C_VEL
LIN {X 0,Y 594.791,Z 123.657,A -85,B 0,C 180,E1 -1147.168,E2 -1147.168} C_VEL
LIN {X 0,Y 594.672,Z 142.749,A -85,B 0,C 180,E1 -1149.776,E2 -1149.776} C_VEL
LIN {X 0,Y 594.575,Z 164.023,A -85,B 0,C 180,E1 -1152.635,E2 -1152.635} C_VEL
LIN {X 0,Y 594.449,Z 183.967,A -85,B 0,C 180,E1 -1155.274,E2 -1155.274} C_VEL
LIN {X 0,Y 594.434,Z 194.438,A -85,B 0,C 180,E1 -1156.649,E2 -1156.649} C_VEL
LIN {X 0,Y 594.75,Z 200.497,A -85,B 0,C 180,E1 -1156.743,E2 -1156.743} C_VEL
LIN {X 0,Y 594.665,Z 302.939,A -85,B 0,C 180,E1 -1157.999,E2 -1157.999} C_VEL
LIN {X 0,Y 594.601,Z 316.214,A -85,B 0,C 180,E1 -1158.3,E2 -1158.3} C_VEL
LIN {X 0,Y 594.599,Z 328.427,A -85,B 0,C 180,E1 -1158.713,E2 -1158.713} C_VEL
LIN {X 0,Y 594.536,Z 340.629,A -85,B 0,C 180,E1 -1159.27,E2 -1159.27} C_VEL
LIN {X 0,Y 594.477,Z 352.199,A -85,B 0,C 180,E1 -1159.957,E2 -1159.957} C_VEL
LIN {X 0,Y 594.414,Z 362.596,A -85,B 0,C 180,E1 -1160.729,E2 -1160.729} C_VEL
LIN {X 0,Y 594.383,Z 371.111,A -85,B 0,C 180,E1 -1161.5,E2 -1161.5} C_VEL
LIN {X 0,Y 594.347,Z 378.959,A -85,B 0,C 180,E1 -1162.355,E2 -1162.355} C_VEL
LIN {X 0,Y 594.283,Z 386.813,A -85,B 0,C 180,E1 -1163.408,E2 -1163.408} C_VEL
LIN {X 0,Y 594.289,Z 393.68,A -85,B 0,C 180,E1 -1164.571,E2 -1164.571} C_VEL
LIN {X 0,Y 594.27,Z 398.371,A -85,B 0,C 180,E1 -1165.591,E2 -1165.591} C_VEL
LIN {X 0,Y 594.267,Z 401.956,A -85,B 0,C 180,E1 -1166.61,E2 -1166.61} C_VEL
LIN {X 0,Y 594.226,Z 403.808,A -85,B 0,C 180,E1 -1167.288,E2 -1167.288} C_VEL
LIN {X 0,Y 594.242,Z 405.2,A -85,B 0,C 180,E1 -1167.967,E2 -1167.967} C_VEL
LIN {X 0,Y 594.239,Z 406.784,A -85,B 0,C 180,E1 -1169.322,E2 -1169.322} C_VEL
LIN {X 0,Y 594.236,Z 407,A -85,B 0,C 180,E1 -1170,E2 -1170} C_VEL
LIN {X 0,Y 594.247,Z 406.185,A -85,B 0,C 180,E1 -1171.355,E2 -1171.355} C_VEL
LIN {X 0,Y 594.242,Z 405.201,A -85,B 0,C 180,E1 -1172.033,E2 -1172.033} C_VEL
LIN {X 0,Y 594.226,Z 403.81,A -85,B 0,C 180,E1 -1172.711,E2 -1172.711} C_VEL
LIN {X 0,Y 594.289,Z 400.896,A -85,B 0,C 180,E1 -1173.729,E2 -1173.729} C_VEL
LIN {X 0,Y 594.241,Z 396.95,A -85,B 0,C 180,E1 -1174.749,E2 -1174.749} C_VEL
LIN {X 0,Y 594.305,Z 390.878,A -85,B 0,C 180,E1 -1175.939,E2 -1175.939} C_VEL
LIN {X 0,Y 594.308,Z 384.237,A -85,B 0,C 180,E1 -1176.962,E2 -1176.962} C_VEL
LIN {X 0,Y 594.359,Z 375.991,A -85,B 0,C 180,E1 -1177.986,E2 -1177.986} C_VEL
LIN {X 0,Y 594.382,Z 367.539,A -85,B 0,C 180,E1 -1178.842,E2 -1178.842} C_VEL
LIN {X 0,Y 594.432,Z 357.096,A -85,B 0,C 180,E1 -1179.699,E2 -1179.699} C_VEL
LIN {X 0,Y 594.481,Z 346.76,A -85,B 0,C 180,E1 -1180.386,E2 -1180.386} C_VEL
LIN {X 0,Y 594.558,Z 335.725,A -85,B 0,C 180,E1 -1180.973,E2 -1180.973} C_VEL
LIN {X 0,Y 594.579,Z 323.715,A -85,B 0,C 180,E1 -1181.464,E2 -1181.464} C_VEL
LIN {X 0,Y 594.648,Z 310.355,A -85,B 0,C 180,E1 -1181.85,E2 -1181.85} C_VEL
LIN {X 0,Y 594.697,Z 297.093,A -85,B 0,C 180,E1 -1182.087,E2 -1182.087} C_VEL
LIN {X 0,Y 594.621,Z 196.047,A -85,B 0,C 180,E1 -1183.314,E2 -1183.314} C_VEL
LIN {X 0,Y 594.415,Z 194.273,A -85,B 0,C 180,E1 -1183.373,E2 -1183.373} C_VEL
LIN {X 0,Y 594.536,Z 172.002,A -85,B 0,C 180,E1 -1186.305,E2 -1186.305} C_VEL
LIN {X 0,Y 594.584,Z 152.785,A -85,B 0,C 180,E1 -1188.871,E2 -1188.871} C_VEL
LIN {X 0,Y 594.769,Z 132.114,A -85,B 0,C 180,E1 -1191.67,E2 -1191.67} C_VEL
LIN {X 0,Y 594.755,Z 121.477,A -85,B 0,C 180,E1 -1193.135,E2 -1193.135} C_VEL
LIN {X 0,Y 594.376,Z 119.447,A -85,B 0,C 180,E1 -1193.45,E2 -1193.45} C_VEL
LIN {X 0,Y 594.386,Z 119.449,A -85,B 0,C 180,E1 -1196.022,E2 -1196.022} C_VEL
LIN {X 0,Y 594.376,Z 119.441,A -85,B 0,C 180,E1 -1198.999,E2 -1198.999} C_VEL
LIN {X 0,Y 594.377,Z 119.445,A -85,B 0,C 180,E1 -1201.642,E2 -1201.642} C_VEL
LIN {X 0,Y 594.374,Z 119.443,A -85,B 0,C 180,E1 -1204.58,E2 -1204.58} C_VEL
LIN {X 0,Y 594.39,Z 119.445,A -85,B 0,C 180,E1 -1207.608,E2 -1207.608} C_VEL
LIN {X 0,Y 594.363,Z 119.443,A -85,B 0,C 180,E1 -1210.567,E2 -1210.567} C_VEL
LIN {X 0,Y 594.367,Z 119.445,A -85,B 0,C 180,E1 -1213.299,E2 -1213.299} C_VEL
LIN {X 0,Y 594.368,Z 119.445,A -85,B 0,C 180,E1 -1216.16,E2 -1216.16} C_VEL
LIN {X 0,Y 594.377,Z 119.441,A -85,B 0,C 180,E1 -1218.536,E2 -1218.536} C_VEL
LIN {X 0,Y 594.382,Z 119.446,A -85,B 0,C 180,E1 -1221.296,E2 -1221.296} C_VEL
LIN {X 0,Y 594.35,Z 119.45,A -85,B 0,C 180,E1 -1223.755,E2 -1223.755} C_VEL
LIN {X 0,Y 594.365,Z 119.443,A -85,B 0,C 180,E1 -1226.238,E2 -1226.238} C_VEL
LIN {X 0,Y 594.369,Z 119.443,A -85,B 0,C 180,E1 -1228.649,E2 -1228.649} C_VEL
LIN {X 0,Y 594.383,Z 119.445,A -85,B 0,C 180,E1 -1231.042,E2 -1231.042} C_VEL
LIN {X 0,Y 594.382,Z 119.451,A -85,B 0,C 180,E1 -1233.3,E2 -1233.3} C_VEL
LIN {X 0,Y 594.381,Z 119.44,A -85,B 0,C 180,E1 -1236.295,E2 -1236.295} C_VEL
LIN {X 0,Y 594.401,Z 119.447,A -85,B 0,C 180,E1 -1239.224,E2 -1239.224} C_VEL
LIN {X 0,Y 594.343,Z 119.445,A -85,B 0,C 180,E1 -1242.094,E2 -1242.094} C_VEL
LIN {X 0,Y 594.362,Z 119.443,A -85,B 0,C 180,E1 -1244.219,E2 -1244.219} C_VEL
LIN {X 0,Y 594.381,Z 119.442,A -85,B 0,C 180,E1 -1246.321,E2 -1246.321} C_VEL
LIN {X 0,Y 594.368,Z 119.45,A -85,B 0,C 180,E1 -1249.094,E2 -1249.094} C_VEL
LIN {X 0,Y 594.381,Z 119.44,A -85,B 0,C 180,E1 -1251.843,E2 -1251.843} C_VEL
LIN {X 0,Y 594.402,Z 119.444,A -85,B 0,C 180,E1 -1254.572,E2 -1254.572} C_VEL
LIN {X 0,Y 594.393,Z 119.441,A -85,B 0,C 180,E1 -1257.289,E2 -1257.289} C_VEL
LIN {X 0,Y 594.414,Z 119.437,A -85,B 0,C 180,E1 -1260,E2 -1260} C_VEL
LIN {X 0,Y 594.409,Z 119.446,A -85,B 0,C 180,E1 -1262.711,E2 -1262.711} C_VEL
LIN {X 0,Y 594.382,Z 119.441,A -85,B 0,C 180,E1 -1265.428,E2 -1265.428} C_VEL
LIN {X 0,Y 594.414,Z 119.441,A -85,B 0,C 180,E1 -1268.157,E2 -1268.157} C_VEL
LIN {X 0,Y 594.387,Z 119.441,A -85,B 0,C 180,E1 -1271.072,E2 -1271.072} C_VEL
LIN {X 0,Y 594.376,Z 119.442,A -85,B 0,C 180,E1 -1273.679,E2 -1273.679} C_VEL
LIN {X 0,Y 594.355,Z 119.444,A -85,B 0,C 180,E1 -1275.328,E2 -1275.328} C_VEL
LIN {X 0,Y 593.682,Z 119.532,A -85,B 0,C 180,E1 -1275.894,E2 -1275.894} C_VEL
LIN {X 0,Y 590.817,Z 119.892,A -85,B 0,C 180,E1 -1276.812,E2 -1276.812} C_VEL
LIN {X 0,Y 588.406,Z 120.195,A -85,B 0,C 180,E1 -1277.551,E2 -1277.551} C_VEL
LIN {X 0,Y 587.382,Z 120.32,A -85,B 0,C 180,E1 -1278.121,E2 -1278.121} C_VEL
LIN {X 0,Y 587.305,Z 120.327,A -85,B 0,C 180,E1 -1278.314,E2 -1278.314} C_VEL
LIN {X 0,Y 587.331,Z 120.319,A -85,B 0,C 180,E1 -1281.037,E2 -1281.037} C_VEL
LIN {X 0,Y 587.314,Z 120.321,A -85,B 0,C 180,E1 -1283.259,E2 -1283.259} C_VEL
LIN {X 0,Y 587.333,Z 120.32,A -85,B 0,C 180,E1 -1285.517,E2 -1285.517} C_VEL
LIN {X 0,Y 587.337,Z 120.324,A -85,B 0,C 180,E1 -1287.818,E2 -1287.818} C_VEL
LIN {X 0,Y 587.335,Z 120.321,A -85,B 0,C 180,E1 -1290.51,E2 -1290.51} C_VEL
LIN {X 0,Y 587.333,Z 120.321,A -85,B 0,C 180,E1 -1293.397,E2 -1293.397} C_VEL
LIN {X 0,Y 587.29,Z 120.334,A -85,B 0,C 180,E1 -1295.9,E2 -1295.9} C_VEL
LIN {X 0,Y 587.323,Z 120.321,A -85,B 0,C 180,E1 -1298.48,E2 -1298.48} C_VEL
LIN {X 0,Y 587.335,Z 120.32,A -85,B 0,C 180,E1 -1301.157,E2 -1301.157} C_VEL
LIN {X 0,Y 587.311,Z 120.325,A -85,B 0,C 180,E1 -1304.112,E2 -1304.112} C_VEL
LIN {X 0,Y 587.316,Z 120.322,A -85,B 0,C 180,E1 -1306.994,E2 -1306.994} C_VEL
LIN {X 0,Y 587.31,Z 120.328,A -85,B 0,C 180,E1 -1309.745,E2 -1309.745} C_VEL
LIN {X 0,Y 587.342,Z 120.317,A -85,B 0,C 180,E1 -1312.392,E2 -1312.392} C_VEL
LIN {X 0,Y 587.342,Z 120.324,A -85,B 0,C 180,E1 -1315.653,E2 -1315.653} C_VEL
LIN {X 0,Y 587.337,Z 120.318,A -85,B 0,C 180,E1 -1318.231,E2 -1318.231} C_VEL
LIN {X 0,Y 587.347,Z 120.32,A -85,B 0,C 180,E1 -1320.867,E2 -1320.867} C_VEL
LIN {X 0,Y 587.337,Z 120.32,A -85,B 0,C 180,E1 -1323.823,E2 -1323.823} C_VEL
LIN {X 0,Y 587.315,Z 120.321,A -85,B 0,C 180,E1 -1325.993,E2 -1325.993} C_VEL
LIN {X 0,Y 587.316,Z 120.321,A -85,B 0,C 180,E1 -1328.226,E2 -1328.226} C_VEL
LIN {X 0,Y 587.343,Z 120.326,A -85,B 0,C 180,E1 -1331.151,E2 -1331.151} C_VEL
LIN {X 0,Y 587.314,Z 120.321,A -85,B 0,C 180,E1 -1334.025,E2 -1334.025} C_VEL
LIN {X 0,Y 587.311,Z 120.33,A -85,B 0,C 180,E1 -1336.858,E2 -1336.858} C_VEL
LIN {X 0,Y 587.337,Z 120.318,A -85,B 0,C 180,E1 -1339.66,E2 -1339.66} C_VEL
LIN {X 0,Y 587.364,Z 120.319,A -85,B 0,C 180,E1 -1342.437,E2 -1342.437} C_VEL
LIN {X 0,Y 587.35,Z 120.32,A -85,B 0,C 180,E1 -1345.195,E2 -1345.195} C_VEL
LIN {X 0,Y 587.373,Z 120.315,A -85,B 0,C 180,E1 -1347.943,E2 -1347.943} C_VEL
LIN {X 0,Y 587.392,Z 120.321,A -85,B 0,C 180,E1 -1350.686,E2 -1350.686} C_VEL
LIN {X 0,Y 587.406,Z 120.467,A -85,B 0,C 180,E1 -1351.8,E2 -1351.8} C_VEL
LIN {X 0,Y 587.355,Z 133.117,A -85,B 0,C 180,E1 -1354.117,E2 -1354.117} C_VEL
LIN {X 0,Y 587.302,Z 146.605,A -85,B 0,C 180,E1 -1356.559,E2 -1356.559} C_VEL
LIN {X 0,Y 587.837,Z 151.277,A -85,B 0,C 180,E1 -1356.639,E2 -1356.639} C_VEL
LIN {X 0,Y 587.659,Z 253.285,A -85,B 0,C 180,E1 -1357.905,E2 -1357.905} C_VEL
LIN {X 0,Y 587.649,Z 267.074,A -85,B 0,C 180,E1 -1358.23,E2 -1358.23} C_VEL
LIN {X 0,Y 587.586,Z 280.028,A -85,B 0,C 180,E1 -1358.685,E2 -1358.685} C_VEL
LIN {X 0,Y 587.529,Z 292.585,A -85,B 0,C 180,E1 -1359.293,E2 -1359.293} C_VEL
LIN {X 0,Y 587.423,Z 303.812,A -85,B 0,C 180,E1 -1359.99,E2 -1359.99} C_VEL
LIN {X 0,Y 587.36,Z 313.948,A -85,B 0,C 180,E1 -1360.776,E2 -1360.776} C_VEL
LIN {X 0,Y 587.296,Z 323.936,A -85,B 0,C 180,E1 -1361.738,E2 -1361.738} C_VEL
LIN {X 0,Y 587.25,Z 332.752,A -85,B 0,C 180,E1 -1362.791,E2 -1362.791} C_VEL
LIN {X 0,Y 587.24,Z 339.792,A -85,B 0,C 180,E1 -1363.849,E2 -1363.849} C_VEL
LIN {X 0,Y 587.204,Z 345.443,A -85,B 0,C 180,E1 -1364.912,E2 -1364.912} C_VEL
LIN {X 0,Y 587.172,Z 349.868,A -85,B 0,C 180,E1 -1365.98,E2 -1365.98} C_VEL
LIN {X 0,Y 587.144,Z 352.368,A -85,B 0,C 180,E1 -1366.748,E2 -1366.748} C_VEL
LIN {X 0,Y 587.132,Z 354.056,A -85,B 0,C 180,E1 -1367.413,E2 -1367.413} C_VEL
LIN {X 0,Y 587.129,Z 355.437,A -85,B 0,C 180,E1 -1368.133,E2 -1368.133} C_VEL
LIN {X 0,Y 587.151,Z 356.526,A -85,B 0,C 180,E1 -1368.985,E2 -1368.985} C_VEL
LIN {X 0,Y 587.123,Z 356.946,A -85,B 0,C 180,E1 -1370.312,E2 -1370.312} C_VEL
LIN {X 0,Y 587.146,Z 356.569,A -85,B 0,C 180,E1 -1371.045,E2 -1371.045} C_VEL
LIN {X 0,Y 587.144,Z 355.718,A -85,B 0,C 180,E1 -1371.781,E2 -1371.781} C_VEL
LIN {X 0,Y 587.147,Z 353.71,A -85,B 0,C 180,E1 -1372.829,E2 -1372.829} C_VEL
LIN {X 0,Y 587.177,Z 350.215,A -85,B 0,C 180,E1 -1374.014,E2 -1374.014} C_VEL
LIN {X 0,Y 587.197,Z 345.605,A -85,B 0,C 180,E1 -1375.144,E2 -1375.144} C_VEL
LIN {X 0,Y 587.243,Z 339.545,A -85,B 0,C 180,E1 -1376.283,E2 -1376.283} C_VEL
LIN {X 0,Y 587.266,Z 333.167,A -85,B 0,C 180,E1 -1377.24,E2 -1377.24} C_VEL
LIN {X 0,Y 587.305,Z 325.282,A -85,B 0,C 180,E1 -1378.208,E2 -1378.208} C_VEL
LIN {X 0,Y 587.362,Z 315.954,A -85,B 0,C 180,E1 -1379.136,E2 -1379.136} C_VEL
LIN {X 0,Y 587.435,Z 305.676,A -85,B 0,C 180,E1 -1379.967,E2 -1379.967} C_VEL
LIN {X 0,Y 587.472,Z 294.178,A -85,B 0,C 180,E1 -1380.709,E2 -1380.709} C_VEL
LIN {X 0,Y 587.598,Z 282.38,A -85,B 0,C 180,E1 -1381.301,E2 -1381.301} C_VEL
LIN {X 0,Y 587.648,Z 270.625,A -85,B 0,C 180,E1 -1381.751,E2 -1381.751} C_VEL
LIN {X 0,Y 587.732,Z 257.888,A -85,B 0,C 180,E1 -1382.095,E2 -1382.095} C_VEL
LIN {X 0,Y 587.749,Z 243.535,A -85,B 0,C 180,E1 -1382.321,E2 -1382.321} C_VEL
LIN {X 0,Y 587.733,Z 149.058,A -85,B 0,C 180,E1 -1383.481,E2 -1383.481} C_VEL
LIN {X 0,Y 587.331,Z 146.631,A -85,B 0,C 180,E1 -1383.525,E2 -1383.525} C_VEL
LIN {X 0,Y 587.39,Z 131.296,A -85,B 0,C 180,E1 -1386.304,E2 -1386.304} C_VEL
LIN {X 0,Y 587.417,Z 121.334,A -85,B 0,C 180,E1 -1388.13,E2 -1388.13} C_VEL
LIN {X 0,Y 587.32,Z 120.324,A -85,B 0,C 180,E1 -1388.352,E2 -1388.352} C_VEL
LIN {X 0,Y 587.334,Z 120.326,A -85,B 0,C 180,E1 -1391.157,E2 -1391.157} C_VEL
LIN {X 0,Y 587.303,Z 120.324,A -85,B 0,C 180,E1 -1394.111,E2 -1394.111} C_VEL
LIN {X 0,Y 587.29,Z 120.331,A -85,B 0,C 180,E1 -1396.991,E2 -1396.991} C_VEL
LIN {X 0,Y 587.301,Z 120.324,A -85,B 0,C 180,E1 -1399.745,E2 -1399.745} C_VEL
LIN {X 0,Y 587.336,Z 120.32,A -85,B 0,C 180,E1 -1402.392,E2 -1402.392} C_VEL
LIN {X 0,Y 587.325,Z 120.321,A -85,B 0,C 180,E1 -1405.656,E2 -1405.656} C_VEL
LIN {X 0,Y 587.315,Z 120.323,A -85,B 0,C 180,E1 -1408.23,E2 -1408.23} C_VEL
LIN {X 0,Y 587.298,Z 120.332,A -85,B 0,C 180,E1 -1410.876,E2 -1410.876} C_VEL
LIN {X 0,Y 587.294,Z 120.324,A -85,B 0,C 180,E1 -1413.832,E2 -1413.832} C_VEL
LIN {X 0,Y 587.284,Z 120.332,A -85,B 0,C 180,E1 -1416.74,E2 -1416.74} C_VEL
LIN {X 0,Y 587.294,Z 120.324,A -85,B 0,C 180,E1 -1419.694,E2 -1419.694} C_VEL
LIN {X 0,Y 587.266,Z 120.334,A -85,B 0,C 180,E1 -1422.592,E2 -1422.592} C_VEL
LIN {X 0,Y 587.302,Z 120.322,A -85,B 0,C 180,E1 -1425.446,E2 -1425.446} C_VEL
LIN {X 0,Y 587.308,Z 120.331,A -85,B 0,C 180,E1 -1428.263,E2 -1428.263} C_VEL
LIN {X 0,Y 587.272,Z 120.326,A -85,B 0,C 180,E1 -1431.05,E2 -1431.05} C_VEL
LIN {X 0,Y 587.306,Z 120.327,A -85,B 0,C 180,E1 -1433.817,E2 -1433.817} C_VEL
LIN {X 0,Y 587.298,Z 120.331,A -85,B 0,C 180,E1 -1435.883,E2 -1435.883} C_VEL
LIN {X 0,Y 587.369,Z 120.323,A -85,B 0,C 180,E1 -1437.943,E2 -1437.943} C_VEL
LIN {X 0,Y 587.38,Z 120.321,A -85,B 0,C 180,E1 -1440,E2 -1440} C_VEL
LIN {X 0,Y 587.332,Z 120.318,A -85,B 0,C 180,E1 -1442.744,E2 -1442.744} C_VEL
LIN {X 0,Y 587.335,Z 120.325,A -85,B 0,C 180,E1 -1445.493,E2 -1445.493} C_VEL
LIN {X 0,Y 587.328,Z 120.32,A -85,B 0,C 180,E1 -1448.256,E2 -1448.256} C_VEL
LIN {X 0,Y 587.333,Z 120.322,A -85,B 0,C 180,E1 -1451.124,E2 -1451.124} C_VEL
LIN {X 0,Y 587.319,Z 120.321,A -85,B 0,C 180,E1 -1454.242,E2 -1454.242} C_VEL
LIN {X 0,Y 587.309,Z 120.324,A -85,B 0,C 180,E1 -1456.8,E2 -1456.8} C_VEL
LIN {X 0,Y 587.302,Z 120.327,A -85,B 0,C 180,E1 -1459.577,E2 -1459.577} C_VEL
LIN {X 0,Y 587.311,Z 120.322,A -85,B 0,C 180,E1 -1461.775,E2 -1461.775} C_VEL
LIN {X 0,Y 587.304,Z 120.327,A -85,B 0,C 180,E1 -1464.761,E2 -1464.761} C_VEL
LIN {X 0,Y 587.329,Z 120.329,A -85,B 0,C 180,E1 -1467.046,E2 -1467.046} C_VEL
LIN {X 0,Y 587.312,Z 120.324,A -85,B 0,C 180,E1 -1469.382,E2 -1469.382} C_VEL
LIN {X 0,Y 587.316,Z 120.321,A -85,B 0,C 180,E1 -1471.831,E2 -1471.831} C_VEL
LIN {X 0,Y 587.338,Z 120.321,A -85,B 0,C 180,E1 -1474.346,E2 -1474.346} C_VEL
LIN {X 0,Y 587.341,Z 120.318,A -85,B 0,C 180,E1 -1477.608,E2 -1477.608} C_VEL
LIN {X 0,Y 587.307,Z 120.326,A -85,B 0,C 180,E1 -1480.255,E2 -1480.255} C_VEL
LIN {X 0,Y 587.306,Z 120.324,A -85,B 0,C 180,E1 -1483.117,E2 -1483.117} C_VEL
LIN {X 0,Y 587.314,Z 120.325,A -85,B 0,C 180,E1 -1486.048,E2 -1486.048} C_VEL
LIN {X 0,Y 587.337,Z 120.321,A -85,B 0,C 180,E1 -1488.925,E2 -1488.925} C_VEL
LIN {X 0,Y 587.324,Z 120.321,A -85,B 0,C 180,E1 -1491.52,E2 -1491.52} C_VEL
LIN {X 0,Y 587.291,Z 120.333,A -85,B 0,C 180,E1 -1494.1,E2 -1494.1} C_VEL
LIN {X 0,Y 587.335,Z 120.322,A -85,B 0,C 180,E1 -1496.603,E2 -1496.603} C_VEL
LIN {X 0,Y 587.325,Z 120.323,A -85,B 0,C 180,E1 -1499.493,E2 -1499.493} C_VEL
LIN {X 0,Y 587.344,Z 120.322,A -85,B 0,C 180,E1 -1502.309,E2 -1502.309} C_VEL
LIN {X 0,Y 587.354,Z 120.319,A -85,B 0,C 180,E1 -1505.241,E2 -1505.241} C_VEL
LIN {X 0,Y 587.365,Z 120.464,A -85,B 0,C 180,E1 -1506.463,E2 -1506.463} C_VEL
LIN {X 0,Y 587.88,Z 126.169,A -85,B 0,C 180,E1 -1507.259,E2 -1507.259} C_VEL
LIN {X 0,Y 587.744,Z 146.738,A -85,B 0,C 180,E1 -1510.075,E2 -1510.075} C_VEL
LIN {X 0,Y 587.57,Z 167.731,A -85,B 0,C 180,E1 -1512.922,E2 -1512.922} C_VEL
LIN {X 0,Y 587.437,Z 188.615,A -85,B 0,C 180,E1 -1515.714,E2 -1515.714} C_VEL
LIN {X 0,Y 587.402,Z 194.438,A -85,B 0,C 180,E1 -1516.486,E2 -1516.486} C_VEL
LIN {X 0,Y 587.84,Z 198.708,A -85,B 0,C 180,E1 -1516.562,E2 -1516.562} C_VEL
LIN {X 0,Y 587.725,Z 302.939,A -85,B 0,C 180,E1 -1517.855,E2 -1517.855} C_VEL
LIN {X 0,Y 587.668,Z 316.215,A -85,B 0,C 180,E1 -1518.16,E2 -1518.16} C_VEL
LIN {X 0,Y 587.629,Z 328.632,A -85,B 0,C 180,E1 -1518.585,E2 -1518.585} C_VEL
LIN {X 0,Y 587.557,Z 340.627,A -85,B 0,C 180,E1 -1519.141,E2 -1519.141} C_VEL
LIN {X 0,Y 587.464,Z 352.201,A -85,B 0,C 180,E1 -1519.836,E2 -1519.836} C_VEL
LIN {X 0,Y 587.366,Z 362.597,A -85,B 0,C 180,E1 -1520.617,E2 -1520.617} C_VEL
LIN {X 0,Y 587.322,Z 371.111,A -85,B 0,C 180,E1 -1521.397,E2 -1521.397} C_VEL
LIN {X 0,Y 587.274,Z 378.959,A -85,B 0,C 180,E1 -1522.263,E2 -1522.263} C_VEL
LIN {X 0,Y 587.23,Z 385.468,A -85,B 0,C 180,E1 -1523.126,E2 -1523.126} C_VEL
LIN {X 0,Y 587.237,Z 391.866,A -85,B 0,C 180,E1 -1524.161,E2 -1524.161} C_VEL
LIN {X 0,Y 587.147,Z 396.949,A -85,B 0,C 180,E1 -1525.194,E2 -1525.194} C_VEL
LIN {X 0,Y 587.213,Z 400.895,A -85,B 0,C 180,E1 -1526.226,E2 -1526.226} C_VEL
LIN {X 0,Y 587.132,Z 403.808,A -85,B 0,C 180,E1 -1527.255,E2 -1527.255} C_VEL
LIN {X 0,Y 587.141,Z 405.199,A -85,B 0,C 180,E1 -1527.942,E2 -1527.942} C_VEL
LIN {X 0,Y 587.14,Z 406.784,A -85,B 0,C 180,E1 -1529.314,E2 -1529.314} C_VEL
LIN {X 0,Y 587.137,Z 407,A -85,B 0,C 180,E1 -1530,E2 -1530} C_VEL
LIN {X 0,Y 587.147,Z 406.186,A -85,B 0,C 180,E1 -1531.372,E2 -1531.372} C_VEL
LIN {X 0,Y 587.141,Z 405.201,A -85,B 0,C 180,E1 -1532.058,E2 -1532.058} C_VEL
LIN {X 0,Y 587.132,Z 403.81,A -85,B 0,C 180,E1 -1532.744,E2 -1532.744} C_VEL
LIN {X 0,Y 587.213,Z 400.896,A -85,B 0,C 180,E1 -1533.774,E2 -1533.774} C_VEL
LIN {X 0,Y 587.147,Z 396.95,A -85,B 0,C 180,E1 -1534.806,E2 -1534.806} C_VEL
LIN {X 0,Y 587.218,Z 390.878,A -85,B 0,C 180,E1 -1536.011,E2 -1536.011} C_VEL
LIN {X 0,Y 587.245,Z 384.238,A -85,B 0,C 180,E1 -1537.046,E2 -1537.046} C_VEL
LIN {X 0,Y 587.299,Z 375.991,A -85,B 0,C 180,E1 -1538.083,E2 -1538.083} C_VEL
LIN {X 0,Y 587.343,Z 367.539,A -85,B 0,C 180,E1 -1538.949,E2 -1538.949} C_VEL
LIN {X 0,Y 587.419,Z 357.098,A -85,B 0,C 180,E1 -1539.816,E2 -1539.816} C_VEL
LIN {X 0,Y 587.497,Z 346.758,A -85,B 0,C 180,E1 -1540.511,E2 -1540.511} C_VEL
LIN {X 0,Y 587.561,Z 334.819,A -85,B 0,C 180,E1 -1541.149,E2 -1541.149} C_VEL
LIN {X 0,Y 587.629,Z 322.602,A -85,B 0,C 180,E1 -1541.639,E2 -1541.639} C_VEL
LIN {X 0,Y 587.703,Z 309.44,A -85,B 0,C 180,E1 -1542.014,E2 -1542.014} C_VEL
LIN {X 0,Y 587.776,Z 297.093,A -85,B 0,C 180,E1 -1542.231,E2 -1542.231} C_VEL
LIN {X 0,Y 587.714,Z 196.716,A -85,B 0,C 180,E1 -1543.465,E2 -1543.465} C_VEL
LIN {X 0,Y 587.401,Z 194.439,A -85,B 0,C 180,E1 -1543.514,E2 -1543.514} C_VEL
LIN {X 0,Y 587.557,Z 173.332,A -85,B 0,C 180,E1 -1546.325,E2 -1546.325} C_VEL
LIN {X 0,Y 587.668,Z 152.571,A -85,B 0,C 180,E1 -1549.131,E2 -1549.131} C_VEL
LIN {X 0,Y 587.873,Z 132.089,A -85,B 0,C 180,E1 -1551.937,E2 -1551.937} C_VEL
LIN {X 0,Y 587.751,Z 122.567,A -85,B 0,C 180,E1 -1553.241,E2 -1553.241} C_VEL
LIN {X 0,Y 587.342,Z 120.325,A -85,B 0,C 180,E1 -1553.585,E2 -1553.585} C_VEL
LIN {X 0,Y 587.339,Z 120.326,A -85,B 0,C 180,E1 -1556.278,E2 -1556.278} C_VEL
LIN {X 0,Y 587.347,Z 120.317,A -85,B 0,C 180,E1 -1559.132,E2 -1559.132} C_VEL
LIN {X 0,Y 587.342,Z 120.325,A -85,B 0,C 180,E1 -1561.835,E2 -1561.835} C_VEL
LIN {X 0,Y 587.345,Z 120.321,A -85,B 0,C 180,E1 -1564.347,E2 -1564.347} C_VEL
LIN {X 0,Y 587.345,Z 120.322,A -85,B 0,C 180,E1 -1567.607,E2 -1567.607} C_VEL
LIN {X 0,Y 587.316,Z 120.324,A -85,B 0,C 180,E1 -1570.254,E2 -1570.254} C_VEL
LIN {X 0,Y 587.314,Z 120.322,A -85,B 0,C 180,E1 -1573.118,E2 -1573.118} C_VEL
LIN {X 0,Y 587.324,Z 120.324,A -85,B 0,C 180,E1 -1576.049,E2 -1576.049} C_VEL
LIN {X 0,Y 587.336,Z 120.319,A -85,B 0,C 180,E1 -1578.925,E2 -1578.925} C_VEL
LIN {X 0,Y 587.328,Z 120.329,A -85,B 0,C 180,E1 -1581.52,E2 -1581.52} C_VEL
LIN {X 0,Y 587.29,Z 120.326,A -85,B 0,C 180,E1 -1584.1,E2 -1584.1} C_VEL
LIN {X 0,Y 587.338,Z 120.32,A -85,B 0,C 180,E1 -1586.888,E2 -1586.888} C_VEL
LIN {X 0,Y 587.326,Z 120.328,A -85,B 0,C 180,E1 -1589.492,E2 -1589.492} C_VEL
LIN {X 0,Y 587.352,Z 120.316,A -85,B 0,C 180,E1 -1592.307,E2 -1592.307} C_VEL
LIN {X 0,Y 587.35,Z 120.327,A -85,B 0,C 180,E1 -1595.241,E2 -1595.241} C_VEL
LIN {X 0,Y 587.317,Z 120.32,A -85,B 0,C 180,E1 -1598.225,E2 -1598.225} C_VEL
LIN {X 0,Y 587.345,Z 120.327,A -85,B 0,C 180,E1 -1601.151,E2 -1601.151} C_VEL
LIN {X 0,Y 587.315,Z 120.321,A -85,B 0,C 180,E1 -1604.024,E2 -1604.024} C_VEL
LIN {X 0,Y 587.359,Z 120.315,A -85,B 0,C 180,E1 -1606.154,E2 -1606.154} C_VEL
LIN {X 0,Y 587.337,Z 120.328,A -85,B 0,C 180,E1 -1608.962,E2 -1608.962} C_VEL
LIN {X 0,Y 587.341,Z 120.318,A -85,B 0,C 180,E1 -1611.744,E2 -1611.744} C_VEL
LIN {X 0,Y 587.367,Z 120.319,A -85,B 0,C 180,E1 -1614.507,E2 -1614.507} C_VEL
LIN {X 0,Y 587.361,Z 120.317,A -85,B 0,C 180,E1 -1617.257,E2 -1617.257} C_VEL
LIN {X 0,Y 587.383,Z 120.313,A -85,B 0,C 180,E1 -1620,E2 -1620} C_VEL
LIN {X 0,Y 587.374,Z 120.322,A -85,B 0,C 180,E1 -1622.743,E2 -1622.743} C_VEL
LIN {X 0,Y 587.351,Z 120.316,A -85,B 0,C 180,E1 -1625.493,E2 -1625.493} C_VEL
LIN {X 0,Y 587.365,Z 120.32,A -85,B 0,C 180,E1 -1628.255,E2 -1628.255} C_VEL
LIN {X 0,Y 587.349,Z 120.317,A -85,B 0,C 180,E1 -1631.134,E2 -1631.134} C_VEL
LIN {X 0,Y 587.365,Z 120.323,A -85,B 0,C 180,E1 -1634.26,E2 -1634.26} C_VEL
LIN {X 0,Y 587.341,Z 120.318,A -85,B 0,C 180,E1 -1637.406,E2 -1637.406} C_VEL
LIN {X 0,Y 587.305,Z 120.327,A -85,B 0,C 180,E1 -1638.314,E2 -1638.314} C_VEL
LIN {X 0,Y 586.662,Z 120.404,A -85,B 0,C 180,E1 -1638.886,E2 -1638.886} C_VEL
LIN {X 0,Y 583.839,Z 120.757,A -85,B 0,C 180,E1 -1639.814,E2 -1639.814} C_VEL
LIN {X 0,Y 581.43,Z 121.058,A -85,B 0,C 180,E1 -1640.561,E2 -1640.561} C_VEL
LIN {X 0,Y 580.377,Z 121.185,A -85,B 0,C 180,E1 -1641.138,E2 -1641.138} C_VEL
LIN {X 0,Y 580.283,Z 121.197,A -85,B 0,C 180,E1 -1641.333,E2 -1641.333} C_VEL
LIN {X 0,Y 580.298,Z 121.202,A -85,B 0,C 180,E1 -1644.316,E2 -1644.316} C_VEL
LIN {X 0,Y 580.274,Z 121.2,A -85,B 0,C 180,E1 -1646.623,E2 -1646.623} C_VEL
LIN {X 0,Y 580.297,Z 121.196,A -85,B 0,C 180,E1 -1649.309,E2 -1649.309} C_VEL
LIN {X 0,Y 580.294,Z 121.201,A -85,B 0,C 180,E1 -1652.201,E2 -1652.201} C_VEL
LIN {X 0,Y 580.286,Z 121.197,A -85,B 0,C 180,E1 -1654.696,E2 -1654.696} C_VEL
LIN {X 0,Y 580.297,Z 121.197,A -85,B 0,C 180,E1 -1657.268,E2 -1657.268} C_VEL
LIN {X 0,Y 580.294,Z 121.198,A -85,B 0,C 180,E1 -1660.271,E2 -1660.271} C_VEL
LIN {X 0,Y 580.275,Z 121.198,A -85,B 0,C 180,E1 -1662.706,E2 -1662.706} C_VEL
LIN {X 0,Y 580.266,Z 121.208,A -85,B 0,C 180,E1 -1665.609,E2 -1665.609} C_VEL
LIN {X 0,Y 580.279,Z 121.199,A -85,B 0,C 180,E1 -1668.231,E2 -1668.231} C_VEL
LIN {X 0,Y 580.277,Z 121.199,A -85,B 0,C 180,E1 -1670.965,E2 -1670.965} C_VEL
LIN {X 0,Y 580.267,Z 121.207,A -85,B 0,C 180,E1 -1673.596,E2 -1673.596} C_VEL
LIN {X 0,Y 580.3,Z 121.195,A -85,B 0,C 180,E1 -1676.144,E2 -1676.144} C_VEL
LIN {X 0,Y 580.272,Z 121.199,A -85,B 0,C 180,E1 -1678.614,E2 -1678.614} C_VEL
LIN {X 0,Y 580.29,Z 121.201,A -85,B 0,C 180,E1 -1681.024,E2 -1681.024} C_VEL
LIN {X 0,Y 580.289,Z 121.199,A -85,B 0,C 180,E1 -1683.667,E2 -1683.667} C_VEL
LIN {X 0,Y 580.291,Z 121.198,A -85,B 0,C 180,E1 -1685.683,E2 -1685.683} C_VEL
LIN {X 0,Y 580.267,Z 121.199,A -85,B 0,C 180,E1 -1687.947,E2 -1687.947} C_VEL
LIN {X 0,Y 580.296,Z 121.203,A -85,B 0,C 180,E1 -1690.913,E2 -1690.913} C_VEL
LIN {X 0,Y 580.264,Z 121.199,A -85,B 0,C 180,E1 -1693.825,E2 -1693.825} C_VEL
LIN {X 0,Y 580.269,Z 121.204,A -85,B 0,C 180,E1 -1696.696,E2 -1696.696} C_VEL
LIN {X 0,Y 580.306,Z 121.203,A -85,B 0,C 180,E1 -1698.827,E2 -1698.827} C_VEL
LIN {X 0,Y 580.309,Z 121.194,A -85,B 0,C 180,E1 -1701.644,E2 -1701.644} C_VEL
LIN {X 0,Y 580.333,Z 121.195,A -85,B 0,C 180,E1 -1704.44,E2 -1704.44} C_VEL
LIN {X 0,Y 580.328,Z 121.194,A -85,B 0,C 180,E1 -1707.224,E2 -1707.224} C_VEL
LIN {X 0,Y 580.353,Z 121.191,A -85,B 0,C 180,E1 -1710,E2 -1710} C_VEL
LIN {X 0,Y 580.366,Z 121.347,A -85,B 0,C 180,E1 -1711.735,E2 -1711.735} C_VEL
LIN {X 0,Y 580.38,Z 132.567,A -85,B 0,C 180,E1 -1713.819,E2 -1713.819} C_VEL
LIN {X 0,Y 580.234,Z 146.599,A -85,B 0,C 180,E1 -1716.391,E2 -1716.391} C_VEL
LIN {X 0,Y 580.924,Z 151.079,A -85,B 0,C 180,E1 -1716.474,E2 -1716.474} C_VEL
LIN {X 0,Y 580.725,Z 253.366,A -85,B 0,C 180,E1 -1717.76,E2 -1717.76} C_VEL
LIN {X 0,Y 580.69,Z 267.149,A -85,B 0,C 180,E1 -1718.088,E2 -1718.088} C_VEL
LIN {X 0,Y 580.641,Z 279.535,A -85,B 0,C 180,E1 -1718.527,E2 -1718.527} C_VEL
LIN {X 0,Y 580.574,Z 290.637,A -85,B 0,C 180,E1 -1719.054,E2 -1719.054} C_VEL
LIN {X 0,Y 580.438,Z 302.238,A -85,B 0,C 180,E1 -1719.76,E2 -1719.76} C_VEL
LIN {X 0,Y 580.358,Z 311.609,A -85,B 0,C 180,E1 -1720.466,E2 -1720.466} C_VEL
LIN {X 0,Y 580.289,Z 321.063,A -85,B 0,C 180,E1 -1721.333,E2 -1721.333} C_VEL
LIN {X 0,Y 580.222,Z 329.163,A -85,B 0,C 180,E1 -1722.238,E2 -1722.238} C_VEL
LIN {X 0,Y 580.133,Z 336.915,A -85,B 0,C 180,E1 -1723.307,E2 -1723.307} C_VEL
LIN {X 0,Y 580.119,Z 343.389,A -85,B 0,C 180,E1 -1724.427,E2 -1724.427} C_VEL
LIN {X 0,Y 580.099,Z 348.085,A -85,B 0,C 180,E1 -1725.458,E2 -1725.458} C_VEL
LIN {X 0,Y 580.075,Z 350.754,A -85,B 0,C 180,E1 -1726.18,E2 -1726.18} C_VEL
LIN {X 0,Y 580.038,Z 352.891,A -85,B 0,C 180,E1 -1726.906,E2 -1726.906} C_VEL
LIN {X 0,Y 580.042,Z 354.579,A -85,B 0,C 180,E1 -1727.633,E2 -1727.633} C_VEL
LIN {X 0,Y 580.037,Z 355.837,A -85,B 0,C 180,E1 -1728.363,E2 -1728.363} C_VEL
LIN {X 0,Y 580.058,Z 356.611,A -85,B 0,C 180,E1 -1729.095,E2 -1729.095} C_VEL
LIN {X 0,Y 580.023,Z 356.959,A -85,B 0,C 180,E1 -1729.833,E2 -1729.833} C_VEL
LIN {X 0,Y 580.043,Z 356.539,A -85,B 0,C 180,E1 -1731.099,E2 -1731.099} C_VEL
LIN {X 0,Y 580.035,Z 355.304,A -85,B 0,C 180,E1 -1732.062,E2 -1732.062} C_VEL
LIN {X 0,Y 580.065,Z 353.473,A -85,B 0,C 180,E1 -1732.956,E2 -1732.956} C_VEL
LIN {X 0,Y 580.088,Z 350.63,A -85,B 0,C 180,E1 -1733.946,E2 -1733.946} C_VEL
LIN {X 0,Y 580.116,Z 346.15,A -85,B 0,C 180,E1 -1735.089,E2 -1735.089} C_VEL
LIN {X 0,Y 580.164,Z 339.842,A -85,B 0,C 180,E1 -1736.308,E2 -1736.308} C_VEL
LIN {X 0,Y 580.208,Z 332.615,A -85,B 0,C 180,E1 -1737.406,E2 -1737.406} C_VEL
LIN {X 0,Y 580.261,Z 324.573,A -85,B 0,C 180,E1 -1738.385,E2 -1738.385} C_VEL
LIN {X 0,Y 580.34,Z 314.631,A -85,B 0,C 180,E1 -1739.366,E2 -1739.366} C_VEL
LIN {X 0,Y 580.396,Z 304.611,A -85,B 0,C 180,E1 -1740.167,E2 -1740.167} C_VEL
LIN {X 0,Y 580.492,Z 292.709,A -85,B 0,C 180,E1 -1740.921,E2 -1740.921} C_VEL
LIN {X 0,Y 580.631,Z 280.615,A -85,B 0,C 180,E1 -1741.517,E2 -1741.517} C_VEL
LIN {X 0,Y 580.718,Z 268.224,A -85,B 0,C 180,E1 -1741.97,E2 -1741.97} C_VEL
LIN {X 0,Y 580.791,Z 254.953,A -85,B 0,C 180,E1 -1742.298,E2 -1742.298} C_VEL
LIN {X 0,Y 580.832,Z 231.656,A -85,B 0,C 180,E1 -1742.617,E2 -1742.617} C_VEL
LIN {X 0,Y 580.899,Z 150.247,A -85,B 0,C 180,E1 -1743.627,E2 -1743.627} C_VEL
LIN {X 0,Y 580.297,Z 146.561,A -85,B 0,C 180,E1 -1743.705,E2 -1743.705} C_VEL
LIN {X 0,Y 580.399,Z 130.406,A -85,B 0,C 180,E1 -1746.67,E2 -1746.67} C_VEL
LIN {X 0,Y 580.294,Z 121.2,A -85,B 0,C 180,E1 -1748.395,E2 -1748.395} C_VEL
LIN {X 0,Y 580.272,Z 121.208,A -85,B 0,C 180,E1 -1751.33,E2 -1751.33} C_VEL
LIN {X 0,Y 580.251,Z 121.202,A -85,B 0,C 180,E1 -1754.389,E2 -1754.389} C_VEL
LIN {X 0,Y 580.254,Z 121.21,A -85,B 0,C 180,E1 -1757.292,E2 -1757.292} C_VEL
LIN {X 0,Y 580.27,Z 121.198,A -85,B 0,C 180,E1 -1760.065,E2 -1760.065} C_VEL
LIN {X 0,Y 580.277,Z 121.206,A -85,B 0,C 180,E1 -1763.069,E2 -1763.069} C_VEL
LIN {X 0,Y 580.27,Z 121.199,A -85,B 0,C 180,E1 -1766.142,E2 -1766.142} C_VEL
LIN {X 0,Y 580.251,Z 121.207,A -85,B 0,C 180,E1 -1768.613,E2 -1768.613} C_VEL
LIN {X 0,Y 580.244,Z 121.208,A -85,B 0,C 180,E1 -1771.021,E2 -1771.021} C_VEL
LIN {X 0,Y 580.25,Z 121.201,A -85,B 0,C 180,E1 -1773.675,E2 -1773.675} C_VEL
LIN {X 0,Y 580.239,Z 121.21,A -85,B 0,C 180,E1 -1776.44,E2 -1776.44} C_VEL
LIN {X 0,Y 580.24,Z 121.203,A -85,B 0,C 180,E1 -1779.436,E2 -1779.436} C_VEL
LIN {X 0,Y 580.232,Z 121.212,A -85,B 0,C 180,E1 -1782.374,E2 -1782.374} C_VEL
LIN {X 0,Y 580.254,Z 121.2,A -85,B 0,C 180,E1 -1785.265,E2 -1785.265} C_VEL
LIN {X 0,Y 580.279,Z 121.205,A -85,B 0,C 180,E1 -1788.118,E2 -1788.118} C_VEL
LIN {X 0,Y 580.232,Z 121.204,A -85,B 0,C 180,E1 -1790.941,E2 -1790.941} C_VEL
LIN {X 0,Y 580.258,Z 121.204,A -85,B 0,C 180,E1 -1793.742,E2 -1793.742} C_VEL
LIN {X 0,Y 580.252,Z 121.208,A -85,B 0,C 180,E1 -1795.833,E2 -1795.833} C_VEL
LIN {X 0,Y 580.338,Z 121.199,A -85,B 0,C 180,E1 -1797.918,E2 -1797.918} C_VEL
LIN {X 0,Y 580.349,Z 121.197,A -85,B 0,C 180,E1 -1800,E2 -1800} C_VEL
LIN {X 0,Y 580.301,Z 121.193,A -85,B 0,C 180,E1 -1802.777,E2 -1802.777} C_VEL
LIN {X 0,Y 580.303,Z 121.202,A -85,B 0,C 180,E1 -1805.56,E2 -1805.56} C_VEL
LIN {X 0,Y 580.295,Z 121.196,A -85,B 0,C 180,E1 -1808.357,E2 -1808.357} C_VEL
LIN {X 0,Y 580.304,Z 121.199,A -85,B 0,C 180,E1 -1811.191,E2 -1811.191} C_VEL
LIN {X 0,Y 580.282,Z 121.197,A -85,B 0,C 180,E1 -1814.324,E2 -1814.324} C_VEL
LIN {X 0,Y 580.269,Z 121.202,A -85,B 0,C 180,E1 -1816.899,E2 -1816.899} C_VEL
LIN {X 0,Y 580.276,Z 121.2,A -85,B 0,C 180,E1 -1819.824,E2 -1819.824} C_VEL
LIN {X 0,Y 580.254,Z 121.2,A -85,B 0,C 180,E1 -1822.054,E2 -1822.054} C_VEL
LIN {X 0,Y 580.282,Z 121.207,A -85,B 0,C 180,E1 -1825.081,E2 -1825.081} C_VEL
LIN {X 0,Y 580.249,Z 121.201,A -85,B 0,C 180,E1 -1827.849,E2 -1827.849} C_VEL
LIN {X 0,Y 580.272,Z 121.204,A -85,B 0,C 180,E1 -1830.692,E2 -1830.692} C_VEL
LIN {X 0,Y 580.281,Z 121.2,A -85,B 0,C 180,E1 -1833.313,E2 -1833.313} C_VEL
LIN {X 0,Y 580.244,Z 121.202,A -85,B 0,C 180,E1 -1835.756,E2 -1835.756} C_VEL
LIN {X 0,Y 580.284,Z 121.199,A -85,B 0,C 180,E1 -1838.147,E2 -1838.147} C_VEL
LIN {X 0,Y 580.296,Z 121.202,A -85,B 0,C 180,E1 -1840.844,E2 -1840.844} C_VEL
LIN {X 0,Y 580.244,Z 121.202,A -85,B 0,C 180,E1 -1843.661,E2 -1843.661} C_VEL
LIN {X 0,Y 580.269,Z 121.206,A -85,B 0,C 180,E1 -1846.61,E2 -1846.61} C_VEL
LIN {X 0,Y 580.299,Z 121.196,A -85,B 0,C 180,E1 -1849.156,E2 -1849.156} C_VEL
LIN {X 0,Y 580.289,Z 121.201,A -85,B 0,C 180,E1 -1851.928,E2 -1851.928} C_VEL
LIN {X 0,Y 580.252,Z 121.206,A -85,B 0,C 180,E1 -1854.453,E2 -1854.453} C_VEL
LIN {X 0,Y 580.291,Z 121.197,A -85,B 0,C 180,E1 -1856.975,E2 -1856.975} C_VEL
LIN {X 0,Y 580.286,Z 121.199,A -85,B 0,C 180,E1 -1859.424,E2 -1859.424} C_VEL
LIN {X 0,Y 580.292,Z 121.204,A -85,B 0,C 180,E1 -1862.143,E2 -1862.143} C_VEL
LIN {X 0,Y 580.308,Z 121.196,A -85,B 0,C 180,E1 -1864.92,E2 -1864.92} C_VEL
LIN {X 0,Y 580.319,Z 121.299,A -85,B 0,C 180,E1 -1866.325,E2 -1866.325} C_VEL
LIN {X 0,Y 580.911,Z 125.765,A -85,B 0,C 180,E1 -1866.964,E2 -1866.964} C_VEL
LIN {X 0,Y 580.819,Z 142.625,A -85,B 0,C 180,E1 -1869.272,E2 -1869.272} C_VEL
LIN {X 0,Y 580.651,Z 162.693,A -85,B 0,C 180,E1 -1872.022,E2 -1872.022} C_VEL
LIN {X 0,Y 580.479,Z 182.637,A -85,B 0,C 180,E1 -1874.732,E2 -1874.732} C_VEL
LIN {X 0,Y 580.408,Z 194.521,A -85,B 0,C 180,E1 -1876.331,E2 -1876.331} C_VEL
LIN {X 0,Y 580.965,Z 200.497,A -85,B 0,C 180,E1 -1876.422,E2 -1876.422} C_VEL
LIN {X 0,Y 580.785,Z 302.939,A -85,B 0,C 180,E1 -1877.708,E2 -1877.708} C_VEL
LIN {X 0,Y 580.742,Z 316.214,A -85,B 0,C 180,E1 -1878.017,E2 -1878.017} C_VEL
LIN {X 0,Y 580.663,Z 327.914,A -85,B 0,C 180,E1 -1878.418,E2 -1878.418} C_VEL
LIN {X 0,Y 580.568,Z 338.929,A -85,B 0,C 180,E1 -1878.92,E2 -1878.92} C_VEL
LIN {X 0,Y 580.461,Z 349.584,A -85,B 0,C 180,E1 -1879.536,E2 -1879.536} C_VEL
LIN {X 0,Y 580.378,Z 360.47,A -85,B 0,C 180,E1 -1880.327,E2 -1880.327} C_VEL
LIN {X 0,Y 580.271,Z 371.111,A -85,B 0,C 180,E1 -1881.292,E2 -1881.292} C_VEL
LIN {X 0,Y 580.222,Z 378.959,A -85,B 0,C 180,E1 -1882.168,E2 -1882.168} C_VEL
LIN {X 0,Y 580.154,Z 386.65,A -85,B 0,C 180,E1 -1883.222,E2 -1883.222} C_VEL
LIN {X 0,Y 580.139,Z 393.679,A -85,B 0,C 180,E1 -1884.438,E2 -1884.438} C_VEL
LIN {X 0,Y 580.108,Z 398.371,A -85,B 0,C 180,E1 -1885.483,E2 -1885.483} C_VEL
LIN {X 0,Y 580.123,Z 401.957,A -85,B 0,C 180,E1 -1886.527,E2 -1886.527} C_VEL
LIN {X 0,Y 580.043,Z 403.808,A -85,B 0,C 180,E1 -1887.222,E2 -1887.222} C_VEL
LIN {X 0,Y 580.04,Z 405.198,A -85,B 0,C 180,E1 -1887.917,E2 -1887.917} C_VEL
LIN {X 0,Y 580.04,Z 406.785,A -85,B 0,C 180,E1 -1889.306,E2 -1889.306} C_VEL
LIN {X 0,Y 580.037,Z 407,A -85,B 0,C 180,E1 -1890,E2 -1890} C_VEL
LIN {X 0,Y 580.047,Z 406.186,A -85,B 0,C 180,E1 -1891.388,E2 -1891.388} C_VEL
LIN {X 0,Y 580.04,Z 405.2,A -85,B 0,C 180,E1 -1892.083,E2 -1892.083} C_VEL
LIN {X 0,Y 580.043,Z 403.81,A -85,B 0,C 180,E1 -1892.778,E2 -1892.778} C_VEL
LIN {X 0,Y 580.11,Z 400.896,A -85,B 0,C 180,E1 -1893.82,E2 -1893.82} C_VEL
LIN {X 0,Y 580.053,Z 396.949,A -85,B 0,C 180,E1 -1894.865,E2 -1894.865} C_VEL
LIN {X 0,Y 580.139,Z 390.877,A -85,B 0,C 180,E1 -1896.085,E2 -1896.085} C_VEL
LIN {X 0,Y 580.184,Z 384.238,A -85,B 0,C 180,E1 -1897.132,E2 -1897.132} C_VEL
LIN {X 0,Y 580.25,Z 375.992,A -85,B 0,C 180,E1 -1898.182,E2 -1898.182} C_VEL
LIN {X 0,Y 580.308,Z 367.54,A -85,B 0,C 180,E1 -1899.058,E2 -1899.058} C_VEL
LIN {X 0,Y 580.422,Z 357.1,A -85,B 0,C 180,E1 -1899.936,E2 -1899.936} C_VEL
LIN {X 0,Y 580.506,Z 346.756,A -85,B 0,C 180,E1 -1900.639,E2 -1900.639} C_VEL
LIN {X 0,Y 580.596,Z 335.249,A -85,B 0,C 180,E1 -1901.264,E2 -1901.264} C_VEL
LIN {X 0,Y 580.682,Z 322.475,A -85,B 0,C 180,E1 -1901.785,E2 -1901.785} C_VEL
LIN {X 0,Y 580.777,Z 309.438,A -85,B 0,C 180,E1 -1902.159,E2 -1902.159} C_VEL
LIN {X 0,Y 580.838,Z 297.093,A -85,B 0,C 180,E1 -1902.38,E2 -1902.38} C_VEL
LIN {X 0,Y 580.802,Z 197.389,A -85,B 0,C 180,E1 -1903.62,E2 -1903.62} C_VEL
LIN {X 0,Y 580.413,Z 194.439,A -85,B 0,C 180,E1 -1903.68,E2 -1903.68} C_VEL
LIN {X 0,Y 580.572,Z 172.002,A -85,B 0,C 180,E1 -1906.708,E2 -1906.708} C_VEL
LIN {X 0,Y 580.727,Z 153.271,A -85,B 0,C 180,E1 -1909.272,E2 -1909.272} C_VEL
LIN {X 0,Y 580.931,Z 133.141,A -85,B 0,C 180,E1 -1912.026,E2 -1912.026} C_VEL
LIN {X 0,Y 580.838,Z 124.036,A -85,B 0,C 180,E1 -1913.287,E2 -1913.287} C_VEL
LIN {X 0,Y 580.296,Z 121.204,A -85,B 0,C 180,E1 -1913.723,E2 -1913.723} C_VEL
LIN {X 0,Y 580.292,Z 121.203,A -85,B 0,C 180,E1 -1916.333,E2 -1916.333} C_VEL
LIN {X 0,Y 580.299,Z 121.196,A -85,B 0,C 180,E1 -1919.309,E2 -1919.309} C_VEL
LIN {X 0,Y 580.297,Z 121.202,A -85,B 0,C 180,E1 -1922.2,E2 -1922.2} C_VEL
LIN {X 0,Y 580.288,Z 121.197,A -85,B 0,C 180,E1 -1924.696,E2 -1924.696} C_VEL
LIN {X 0,Y 580.3,Z 121.196,A -85,B 0,C 180,E1 -1927.268,E2 -1927.268} C_VEL
LIN {X 0,Y 580.296,Z 121.198,A -85,B 0,C 180,E1 -1930.271,E2 -1930.271} C_VEL
LIN {X 0,Y 580.277,Z 121.197,A -85,B 0,C 180,E1 -1932.706,E2 -1932.706} C_VEL
LIN {X 0,Y 580.268,Z 121.207,A -85,B 0,C 180,E1 -1935.609,E2 -1935.609} C_VEL
LIN {X 0,Y 580.281,Z 121.199,A -85,B 0,C 180,E1 -1938.231,E2 -1938.231} C_VEL
LIN {X 0,Y 580.278,Z 121.199,A -85,B 0,C 180,E1 -1940.965,E2 -1940.965} C_VEL
LIN {X 0,Y 580.269,Z 121.207,A -85,B 0,C 180,E1 -1943.596,E2 -1943.596} C_VEL
LIN {X 0,Y 580.301,Z 121.195,A -85,B 0,C 180,E1 -1946.144,E2 -1946.144} C_VEL
LIN {X 0,Y 580.273,Z 121.198,A -85,B 0,C 180,E1 -1948.614,E2 -1948.614} C_VEL
LIN {X 0,Y 580.292,Z 121.2,A -85,B 0,C 180,E1 -1951.024,E2 -1951.024} C_VEL
LIN {X 0,Y 580.29,Z 121.2,A -85,B 0,C 180,E1 -1953.666,E2 -1953.666} C_VEL
LIN {X 0,Y 580.295,Z 121.198,A -85,B 0,C 180,E1 -1955.683,E2 -1955.683} C_VEL
LIN {X 0,Y 580.269,Z 121.199,A -85,B 0,C 180,E1 -1957.947,E2 -1957.947} C_VEL
LIN {X 0,Y 580.297,Z 121.201,A -85,B 0,C 180,E1 -1960.913,E2 -1960.913} C_VEL
LIN {X 0,Y 580.265,Z 121.199,A -85,B 0,C 180,E1 -1963.825,E2 -1963.825} C_VEL
LIN {X 0,Y 580.326,Z 121.191,A -85,B 0,C 180,E1 -1965.983,E2 -1965.983} C_VEL
LIN {X 0,Y 580.306,Z 121.202,A -85,B 0,C 180,E1 -1968.827,E2 -1968.827} C_VEL
LIN {X 0,Y 580.31,Z 121.194,A -85,B 0,C 180,E1 -1971.643,E2 -1971.643} C_VEL
LIN {X 0,Y 580.332,Z 121.195,A -85,B 0,C 180,E1 -1974.44,E2 -1974.44} C_VEL
LIN {X 0,Y 580.329,Z 121.194,A -85,B 0,C 180,E1 -1977.223,E2 -1977.223} C_VEL
LIN {X 0,Y 580.353,Z 121.189,A -85,B 0,C 180,E1 -1980,E2 -1980} C_VEL
LIN {X 0,Y 580.34,Z 121.197,A -85,B 0,C 180,E1 -1982.776,E2 -1982.776} C_VEL
LIN {X 0,Y 580.32,Z 121.192,A -85,B 0,C 180,E1 -1985.56,E2 -1985.56} C_VEL
LIN {X 0,Y 580.328,Z 121.199,A -85,B 0,C 180,E1 -1988.356,E2 -1988.356} C_VEL
LIN {X 0,Y 580.3,Z 121.195,A -85,B 0,C 180,E1 -1991.191,E2 -1991.191} C_VEL
LIN {X 0,Y 580.324,Z 121.196,A -85,B 0,C 180,E1 -1994.017,E2 -1994.017} C_VEL
LIN {X 0,Y 580.313,Z 121.195,A -85,B 0,C 180,E1 -1996.914,E2 -1996.914} C_VEL
LIN {X 0,Y 580.286,Z 121.2,A -85,B 0,C 180,E1 -1999.823,E2 -1999.823} C_VEL
LIN {X 0,Y 580.283,Z 121.197,A -85,B 0,C 180,E1 -2001.333,E2 -2001.333} C_VEL
LIN {X 0,Y 579.585,Z 121.291,A -85,B 0,C 180,E1 -2001.912,E2 -2001.912} C_VEL
LIN {X 0,Y 576.707,Z 121.645,A -85,B 0,C 180,E1 -2002.852,E2 -2002.852} C_VEL
LIN {X 0,Y 574.312,Z 121.943,A -85,B 0,C 180,E1 -2003.608,E2 -2003.608} C_VEL
LIN {X 0,Y 573.314,Z 122.074,A -85,B 0,C 180,E1 -2004.192,E2 -2004.192} C_VEL
LIN {X 0,Y 573.248,Z 122.075,A -85,B 0,C 180,E1 -2004.39,E2 -2004.39} C_VEL
LIN {X 0,Y 573.218,Z 122.077,A -85,B 0,C 180,E1 -2006.977,E2 -2006.977} C_VEL
LIN {X 0,Y 573.243,Z 122.076,A -85,B 0,C 180,E1 -2009.488,E2 -2009.488} C_VEL
LIN {X 0,Y 573.251,Z 122.074,A -85,B 0,C 180,E1 -2012.645,E2 -2012.645} C_VEL
LIN {X 0,Y 573.205,Z 122.079,A -85,B 0,C 180,E1 -2015.188,E2 -2015.188} C_VEL
LIN {X 0,Y 573.234,Z 122.085,A -85,B 0,C 180,E1 -2017.808,E2 -2017.808} C_VEL
LIN {X 0,Y 573.244,Z 122.074,A -85,B 0,C 180,E1 -2020.525,E2 -2020.525} C_VEL
LIN {X 0,Y 573.235,Z 122.079,A -85,B 0,C 180,E1 -2023.359,E2 -2023.359} C_VEL
LIN {X 0,Y 573.244,Z 122.075,A -85,B 0,C 180,E1 -2026.331,E2 -2026.331} C_VEL
LIN {X 0,Y 573.228,Z 122.076,A -85,B 0,C 180,E1 -2028.543,E2 -2028.543} C_VEL
LIN {X 0,Y 573.241,Z 122.08,A -85,B 0,C 180,E1 -2031.298,E2 -2031.298} C_VEL
LIN {X 0,Y 573.212,Z 122.08,A -85,B 0,C 180,E1 -2034.019,E2 -2034.019} C_VEL
LIN {X 0,Y 573.238,Z 122.074,A -85,B 0,C 180,E1 -2036.516,E2 -2036.516} C_VEL
LIN {X 0,Y 573.223,Z 122.082,A -85,B 0,C 180,E1 -2039.119,E2 -2039.119} C_VEL
LIN {X 0,Y 573.235,Z 122.082,A -85,B 0,C 180,E1 -2041.436,E2 -2041.436} C_VEL
LIN {X 0,Y 573.259,Z 122.074,A -85,B 0,C 180,E1 -2043.81,E2 -2043.81} C_VEL
LIN {X 0,Y 573.222,Z 122.076,A -85,B 0,C 180,E1 -2046.134,E2 -2046.134} C_VEL
LIN {X 0,Y 573.248,Z 122.082,A -85,B 0,C 180,E1 -2049.174,E2 -2049.174} C_VEL
LIN {X 0,Y 573.214,Z 122.082,A -85,B 0,C 180,E1 -2051.411,E2 -2051.411} C_VEL
LIN {X 0,Y 573.239,Z 122.076,A -85,B 0,C 180,E1 -2053.622,E2 -2053.622} C_VEL
LIN {X 0,Y 573.227,Z 122.079,A -85,B 0,C 180,E1 -2056.529,E2 -2056.529} C_VEL
LIN {X 0,Y 573.264,Z 122.079,A -85,B 0,C 180,E1 -2058.745,E2 -2058.745} C_VEL
LIN {X 0,Y 573.254,Z 122.073,A -85,B 0,C 180,E1 -2061.54,E2 -2061.54} C_VEL
LIN {X 0,Y 573.299,Z 122.071,A -85,B 0,C 180,E1 -2064.372,E2 -2064.372} C_VEL
LIN {X 0,Y 573.313,Z 122.066,A -85,B 0,C 180,E1 -2067.893,E2 -2067.893} C_VEL
LIN {X 0,Y 573.333,Z 122.073,A -85,B 0,C 180,E1 -2070.702,E2 -2070.702} C_VEL
LIN {X 0,Y 573.297,Z 122.19,A -85,B 0,C 180,E1 -2071.669,E2 -2071.669} C_VEL
LIN {X 0,Y 573.333,Z 132.036,A -85,B 0,C 180,E1 -2073.514,E2 -2073.514} C_VEL
LIN {X 0,Y 573.188,Z 146.271,A -85,B 0,C 180,E1 -2076.159,E2 -2076.159} C_VEL
LIN {X 0,Y 573.197,Z 146.627,A -85,B 0,C 180,E1 -2076.225,E2 -2076.225} C_VEL
LIN {X 0,Y 574.041,Z 152.54,A -85,B 0,C 180,E1 -2076.326,E2 -2076.326} C_VEL
LIN {X 0,Y 573.804,Z 253.423,A -85,B 0,C 180,E1 -2077.61,E2 -2077.61} C_VEL
LIN {X 0,Y 573.754,Z 267.198,A -85,B 0,C 180,E1 -2077.943,E2 -2077.943} C_VEL
LIN {X 0,Y 573.667,Z 280.107,A -85,B 0,C 180,E1 -2078.41,E2 -2078.41} C_VEL
LIN {X 0,Y 573.584,Z 291.858,A -85,B 0,C 180,E1 -2078.988,E2 -2078.988} C_VEL
LIN {X 0,Y 573.422,Z 303.242,A -85,B 0,C 180,E1 -2079.702,E2 -2079.702} C_VEL
LIN {X 0,Y 573.301,Z 313.507,A -85,B 0,C 180,E1 -2080.507,E2 -2080.507} C_VEL
LIN {X 0,Y 573.21,Z 323.571,A -85,B 0,C 180,E1 -2081.493,E2 -2081.493} C_VEL
LIN {X 0,Y 573.157,Z 332.455,A -85,B 0,C 180,E1 -2082.571,E2 -2082.571} C_VEL
LIN {X 0,Y 573.078,Z 339.565,A -85,B 0,C 180,E1 -2083.655,E2 -2083.655} C_VEL
LIN {X 0,Y 573.031,Z 346.087,A -85,B 0,C 180,E1 -2084.925,E2 -2084.925} C_VEL
LIN {X 0,Y 572.996,Z 350.364,A -85,B 0,C 180,E1 -2086.02,E2 -2086.02} C_VEL
LIN {X 0,Y 572.938,Z 353.535,A -85,B 0,C 180,E1 -2087.122,E2 -2087.122} C_VEL
LIN {X 0,Y 572.944,Z 355.074,A -85,B 0,C 180,E1 -2087.858,E2 -2087.858} C_VEL
LIN {X 0,Y 572.967,Z 356.678,A -85,B 0,C 180,E1 -2089.182,E2 -2089.182} C_VEL
LIN {X 0,Y 572.949,Z 356.996,A -85,B 0,C 180,E1 -2090.088,E2 -2090.088} C_VEL
LIN {X 0,Y 572.964,Z 356.445,A -85,B 0,C 180,E1 -2091.217,E2 -2091.217} C_VEL
LIN {X 0,Y 572.945,Z 354.858,A -85,B 0,C 180,E1 -2092.35,E2 -2092.35} C_VEL
LIN {X 0,Y 572.979,Z 352.162,A -85,B 0,C 180,E1 -2093.493,E2 -2093.493} C_VEL
LIN {X 0,Y 573.014,Z 347.543,A -85,B 0,C 180,E1 -2094.823,E2 -2094.823} C_VEL
LIN {X 0,Y 573.063,Z 341.994,A -85,B 0,C 180,E1 -2096.004,E2 -2096.004} C_VEL
LIN {X 0,Y 573.111,Z 334.83,A -85,B 0,C 180,E1 -2097.18,E2 -2097.18} C_VEL
LIN {X 0,Y 573.192,Z 326.6,A -85,B 0,C 180,E1 -2098.256,E2 -2098.256} C_VEL
LIN {X 0,Y 573.264,Z 318.063,A -85,B 0,C 180,E1 -2099.165,E2 -2099.165} C_VEL
LIN {X 0,Y 573.368,Z 308.682,A -85,B 0,C 180,E1 -2099.983,E2 -2099.983} C_VEL
LIN {X 0,Y 573.472,Z 297.424,A -85,B 0,C 180,E1 -2100.774,E2 -2100.774} C_VEL
LIN {X 0,Y 573.633,Z 285.578,A -85,B 0,C 180,E1 -2101.431,E2 -2101.431} C_VEL
LIN {X 0,Y 573.75,Z 273.131,A -85,B 0,C 180,E1 -2101.952,E2 -2101.952} C_VEL
LIN {X 0,Y 573.841,Z 259.948,A -85,B 0,C 180,E1 -2102.341,E2 -2102.341} C_VEL
LIN {X 0,Y 573.884,Z 246.755,A -85,B 0,C 180,E1 -2102.582,E2 -2102.582} C_VEL
LIN {X 0,Y 574.029,Z 151.284,A -85,B 0,C 180,E1 -2103.78,E2 -2103.78} C_VEL
LIN {X 0,Y 573.251,Z 146.587,A -85,B 0,C 180,E1 -2103.871,E2 -2103.871} C_VEL
LIN {X 0,Y 573.369,Z 131.404,A -85,B 0,C 180,E1 -2106.695,E2 -2106.695} C_VEL
LIN {X 0,Y 573.268,Z 122.075,A -85,B 0,C 180,E1 -2108.44,E2 -2108.44} C_VEL
LIN {X 0,Y 573.218,Z 122.086,A -85,B 0,C 180,E1 -2111.458,E2 -2111.458} C_VEL
LIN {X 0,Y 573.217,Z 122.079,A -85,B 0,C 180,E1 -2114.335,E2 -2114.335} C_VEL
LIN {X 0,Y 573.217,Z 122.086,A -85,B 0,C 180,E1 -2117.361,E2 -2117.361} C_VEL
LIN {X 0,Y 573.23,Z 122.076,A -85,B 0,C 180,E1 -2120.392,E2 -2120.392} C_VEL
LIN {X 0,Y 573.231,Z 122.083,A -85,B 0,C 180,E1 -2123.076,E2 -2123.076} C_VEL
LIN {X 0,Y 573.245,Z 122.075,A -85,B 0,C 180,E1 -2125.67,E2 -2125.67} C_VEL
LIN {X 0,Y 573.22,Z 122.078,A -85,B 0,C 180,E1 -2128.183,E2 -2128.183} C_VEL
LIN {X 0,Y 573.214,Z 122.085,A -85,B 0,C 180,E1 -2130.631,E2 -2130.631} C_VEL
LIN {X 0,Y 573.197,Z 122.08,A -85,B 0,C 180,E1 -2133.516,E2 -2133.516} C_VEL
LIN {X 0,Y 573.19,Z 122.084,A -85,B 0,C 180,E1 -2136.133,E2 -2136.133} C_VEL
LIN {X 0,Y 573.216,Z 122.079,A -85,B 0,C 180,E1 -2139.172,E2 -2139.172} C_VEL
LIN {X 0,Y 573.193,Z 122.085,A -85,B 0,C 180,E1 -2142.15,E2 -2142.15} C_VEL
LIN {X 0,Y 573.203,Z 122.079,A -85,B 0,C 180,E1 -2145.08,E2 -2145.08} C_VEL
LIN {X 0,Y 573.221,Z 122.082,A -85,B 0,C 180,E1 -2147.97,E2 -2147.97} C_VEL
LIN {X 0,Y 573.198,Z 122.087,A -85,B 0,C 180,E1 -2150.116,E2 -2150.116} C_VEL
LIN {X 0,Y 573.22,Z 122.076,A -85,B 0,C 180,E1 -2152.958,E2 -2152.958} C_VEL
LIN {X 0,Y 573.269,Z 122.07,A -85,B 0,C 180,E1 -2155.077,E2 -2155.077} C_VEL
LIN {X 0,Y 573.308,Z 122.074,A -85,B 0,C 180,E1 -2157.893,E2 -2157.893} C_VEL
LIN {X 0,Y 573.317,Z 122.072,A -85,B 0,C 180,E1 -2160,E2 -2160} C_VEL
LIN {X 0,Y 573.269,Z 122.069,A -85,B 0,C 180,E1 -2162.811,E2 -2162.811} C_VEL
LIN {X 0,Y 573.271,Z 122.079,A -85,B 0,C 180,E1 -2165.629,E2 -2165.629} C_VEL
LIN {X 0,Y 573.236,Z 122.074,A -85,B 0,C 180,E1 -2168.46,E2 -2168.46} C_VEL
LIN {X 0,Y 573.274,Z 122.077,A -85,B 0,C 180,E1 -2171.312,E2 -2171.312} C_VEL
LIN {X 0,Y 573.259,Z 122.072,A -85,B 0,C 180,E1 -2174.414,E2 -2174.414} C_VEL
LIN {X 0,Y 573.239,Z 122.08,A -85,B 0,C 180,E1 -2177.112,E2 -2177.112} C_VEL
LIN {X 0,Y 573.232,Z 122.076,A -85,B 0,C 180,E1 -2180.078,E2 -2180.078} C_VEL
LIN {X 0,Y 573.221,Z 122.075,A -85,B 0,C 180,E1 -2182.339,E2 -2182.339} C_VEL
LIN {X 0,Y 573.236,Z 122.079,A -85,B 0,C 180,E1 -2185.411,E2 -2185.411} C_VEL
LIN {X 0,Y 573.205,Z 122.079,A -85,B 0,C 180,E1 -2188.02,E2 -2188.02} C_VEL
LIN {X 0,Y 573.23,Z 122.076,A -85,B 0,C 180,E1 -2190.177,E2 -2190.177} C_VEL
LIN {X 0,Y 573.248,Z 122.08,A -85,B 0,C 180,E1 -2192.646,E2 -2192.646} C_VEL
LIN {X 0,Y 573.206,Z 122.082,A -85,B 0,C 180,E1 -2195.188,E2 -2195.188} C_VEL
LIN {X 0,Y 573.232,Z 122.075,A -85,B 0,C 180,E1 -2197.808,E2 -2197.808} C_VEL
LIN {X 0,Y 573.247,Z 122.082,A -85,B 0,C 180,E1 -2200.525,E2 -2200.525} C_VEL
LIN {X 0,Y 573.211,Z 122.079,A -85,B 0,C 180,E1 -2203.362,E2 -2203.362} C_VEL
LIN {X 0,Y 573.238,Z 122.083,A -85,B 0,C 180,E1 -2206.332,E2 -2206.332} C_VEL
LIN {X 0,Y 573.248,Z 122.074,A -85,B 0,C 180,E1 -2209.475,E2 -2209.475} C_VEL
LIN {X 0,Y 573.233,Z 122.084,A -85,B 0,C 180,E1 -2212.192,E2 -2212.192} C_VEL
LIN {X 0,Y 573.235,Z 122.075,A -85,B 0,C 180,E1 -2215.229,E2 -2215.229} C_VEL
LIN {X 0,Y 573.25,Z 122.079,A -85,B 0,C 180,E1 -2217.773,E2 -2217.773} C_VEL
LIN {X 0,Y 573.246,Z 122.076,A -85,B 0,C 180,E1 -2220.633,E2 -2220.633} C_VEL
LIN {X 0,Y 573.221,Z 122.078,A -85,B 0,C 180,E1 -2223.022,E2 -2223.022} C_VEL
LIN {X 0,Y 573.278,Z 122.075,A -85,B 0,C 180,E1 -2225.366,E2 -2225.366} C_VEL
LIN {X 0,Y 573.265,Z 122.11,A -85,B 0,C 180,E1 -2226.181,E2 -2226.181} C_VEL
LIN {X 0,Y 573.962,Z 127.287,A -85,B 0,C 180,E1 -2226.931,E2 -2226.931} C_VEL
LIN {X 0,Y 573.824,Z 144.995,A -85,B 0,C 180,E1 -2229.383,E2 -2229.383} C_VEL
LIN {X 0,Y 573.658,Z 166.815,A -85,B 0,C 180,E1 -2232.367,E2 -2232.367} C_VEL
LIN {X 0,Y 573.451,Z 186.626,A -85,B 0,C 180,E1 -2235.086,E2 -2235.086} C_VEL
LIN {X 0,Y 573.412,Z 194.521,A -85,B 0,C 180,E1 -2236.161,E2 -2236.161} C_VEL
LIN {X 0,Y 574.059,Z 200.497,A -85,B 0,C 180,E1 -2236.256,E2 -2236.256} C_VEL
LIN {X 0,Y 573.85,Z 302.939,A -85,B 0,C 180,E1 -2237.557,E2 -2237.557} C_VEL
LIN {X 0,Y 573.803,Z 316.213,A -85,B 0,C 180,E1 -2237.87,E2 -2237.87} C_VEL
LIN {X 0,Y 573.7,Z 328.373,A -85,B 0,C 180,E1 -2238.294,E2 -2238.294} C_VEL
LIN {X 0,Y 573.566,Z 340.623,A -85,B 0,C 180,E1 -2238.873,E2 -2238.873} C_VEL
LIN {X 0,Y 573.428,Z 352.196,A -85,B 0,C 180,E1 -2239.585,E2 -2239.585} C_VEL
LIN {X 0,Y 573.333,Z 362.601,A -85,B 0,C 180,E1 -2240.385,E2 -2240.385} C_VEL
LIN {X 0,Y 573.241,Z 371.111,A -85,B 0,C 180,E1 -2241.184,E2 -2241.184} C_VEL
LIN {X 0,Y 573.161,Z 378.959,A -85,B 0,C 180,E1 -2242.071,E2 -2242.071} C_VEL
LIN {X 0,Y 573.073,Z 386.581,A -85,B 0,C 180,E1 -2243.126,E2 -2243.126} C_VEL
LIN {X 0,Y 573.071,Z 393.679,A -85,B 0,C 180,E1 -2244.37,E2 -2244.37} C_VEL
LIN {X 0,Y 573.028,Z 398.372,A -85,B 0,C 180,E1 -2245.427,E2 -2245.427} C_VEL
LIN {X 0,Y 573.022,Z 401.957,A -85,B 0,C 180,E1 -2246.484,E2 -2246.484} C_VEL
LIN {X 0,Y 572.959,Z 403.808,A -85,B 0,C 180,E1 -2247.188,E2 -2247.188} C_VEL
LIN {X 0,Y 572.946,Z 406.185,A -85,B 0,C 180,E1 -2248.594,E2 -2248.594} C_VEL
LIN {X 0,Y 572.938,Z 407,A -85,B 0,C 180,E1 -2250,E2 -2250} C_VEL
LIN {X 0,Y 572.946,Z 406.186,A -85,B 0,C 180,E1 -2251.406,E2 -2251.406} C_VEL
LIN {X 0,Y 572.94,Z 405.199,A -85,B 0,C 180,E1 -2252.109,E2 -2252.109} C_VEL
LIN {X 0,Y 572.959,Z 403.81,A -85,B 0,C 180,E1 -2252.812,E2 -2252.812} C_VEL
LIN {X 0,Y 573.015,Z 400.896,A -85,B 0,C 180,E1 -2253.868,E2 -2253.868} C_VEL
LIN {X 0,Y 572.963,Z 396.949,A -85,B 0,C 180,E1 -2254.925,E2 -2254.925} C_VEL
LIN {X 0,Y 573.065,Z 390.877,A -85,B 0,C 180,E1 -2256.16,E2 -2256.16} C_VEL
LIN {X 0,Y 573.119,Z 384.238,A -85,B 0,C 180,E1 -2257.221,E2 -2257.221} C_VEL
LIN {X 0,Y 573.201,Z 375.992,A -85,B 0,C 180,E1 -2258.283,E2 -2258.283} C_VEL
LIN {X 0,Y 573.287,Z 367.54,A -85,B 0,C 180,E1 -2259.17,E2 -2259.17} C_VEL
LIN {X 0,Y 573.427,Z 357.097,A -85,B 0,C 180,E1 -2260.058,E2 -2260.058} C_VEL
LIN {X 0,Y 573.543,Z 345.433,A -85,B 0,C 180,E1 -2260.853,E2 -2260.853} C_VEL
LIN {X 0,Y 573.651,Z 334.31,A -85,B 0,C 180,E1 -2261.446,E2 -2261.446} C_VEL
LIN {X 0,Y 573.745,Z 321.173,A -85,B 0,C 180,E1 -2261.974,E2 -2261.974} C_VEL
LIN {X 0,Y 573.871,Z 308.522,A -85,B 0,C 180,E1 -2262.33,E2 -2262.33} C_VEL
LIN {X 0,Y 573.938,Z 295.319,A -85,B 0,C 180,E1 -2262.553,E2 -2262.553} C_VEL
LIN {X 0,Y 573.907,Z 198.06,A -85,B 0,C 180,E1 -2263.779,E2 -2263.779} C_VEL
LIN {X 0,Y 573.417,Z 194.439,A -85,B 0,C 180,E1 -2263.85,E2 -2263.85} C_VEL
